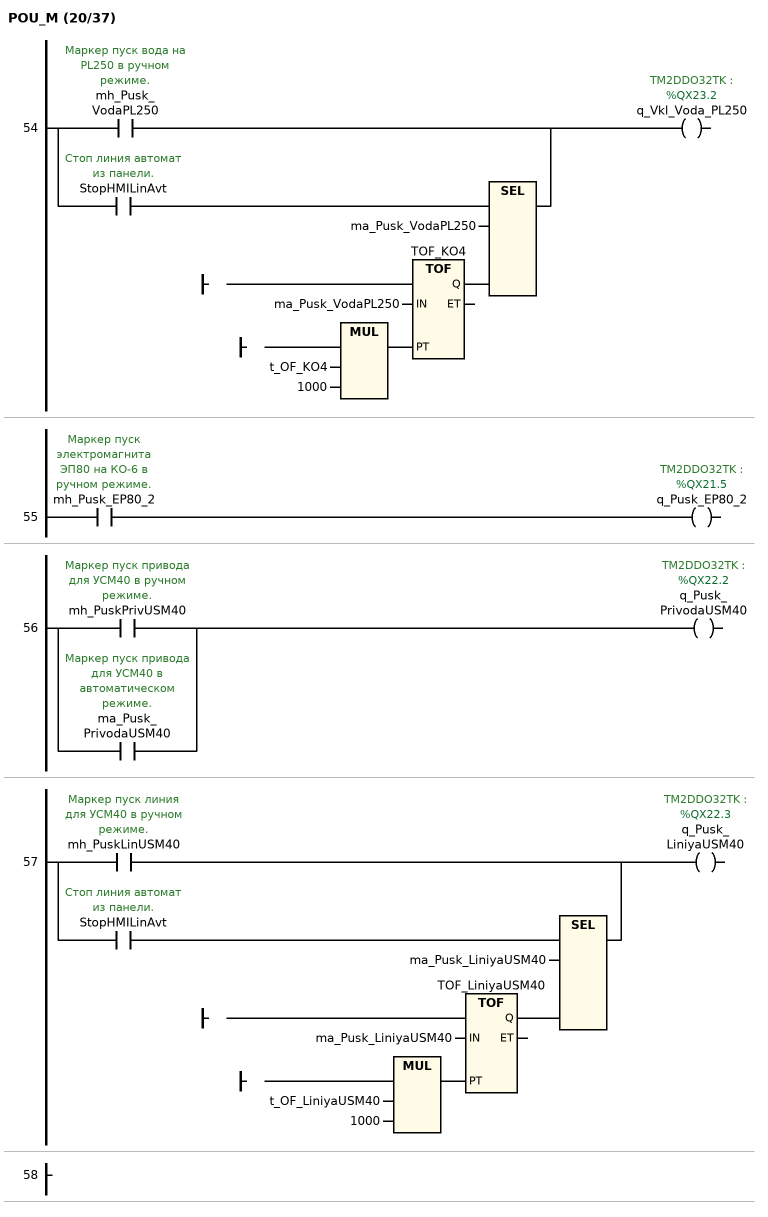
// NETWORK 54
//   mh_Pusk_VodaPL250: Маркер пуск вода на PL250 в ручном режиме.
//   StopHMILinAvt: Стоп линия автомат из панели.
//   ma_Pusk_VodaPL250: Маркер включение воды в питатель PL250 в автоматическом режиме.
//   TOF_KO4: Задержка перед выключением КО-4 при "Стоп линия автомат".
//   t_OF_KO4: Время задержки перед выключением КО-4 при Стоп Линия Автомат.
//   q_Vkl_Voda_PL250: TM2DDO32TK : | AT %QX23.2
TOF_KO4(IN := ma_Pusk_VodaPL250, PT := t_OF_KO4 * 1000); // TOF
q_Vkl_Voda_PL250 := mh_Pusk_VodaPL250 OR SEL(StopHMILinAvt, ma_Pusk_VodaPL250, TOF_KO4.Q);

// NETWORK 55
//   mh_Pusk_EP80_2: Маркер пуск электромагнита ЭП80 на КО-6 в ручном режиме.
//   q_Pusk_EP80_2: TM2DDO32TK : | AT %QX21.5
q_Pusk_EP80_2 := mh_Pusk_EP80_2;

// NETWORK 56
//   mh_PuskPrivUSM40: Маркер пуск привода для УСМ40 в ручном режиме.
//   ma_Pusk_PrivodaUSM40: Маркер пуск привода для УСМ40 в автоматическом режиме.
//   q_Pusk_PrivodaUSM40: TM2DDO32TK : | AT %QX22.2
q_Pusk_PrivodaUSM40 := mh_PuskPrivUSM40 OR ma_Pusk_PrivodaUSM40;

// NETWORK 57
//   mh_PuskLinUSM40: Маркер пуск линия для УСМ40 в ручном режиме.
//   StopHMILinAvt: Стоп линия автомат из панели.
//   ma_Pusk_LiniyaUSM40: Маркер пуск линия для УСМ40 в автоматическом режиме.
//   TOF_LiniyaUSM40: Задержка перед выключением конвейера на УСМ40 при "Стоп линия автомат".
//   t_OF_LiniyaUSM40: Время задержки перед выключением линии на УСМ40 при Стоп Линия Автомат.
//   q_Pusk_LiniyaUSM40: TM2DDO32TK : | AT %QX22.3
TOF_LiniyaUSM40(IN := ma_Pusk_LiniyaUSM40, PT := t_OF_LiniyaUSM40 * 1000); // TOF
q_Pusk_LiniyaUSM40 := mh_PuskLinUSM40 OR SEL(StopHMILinAvt, ma_Pusk_LiniyaUSM40, TOF_LiniyaUSM40.Q);

// NETWORK 58

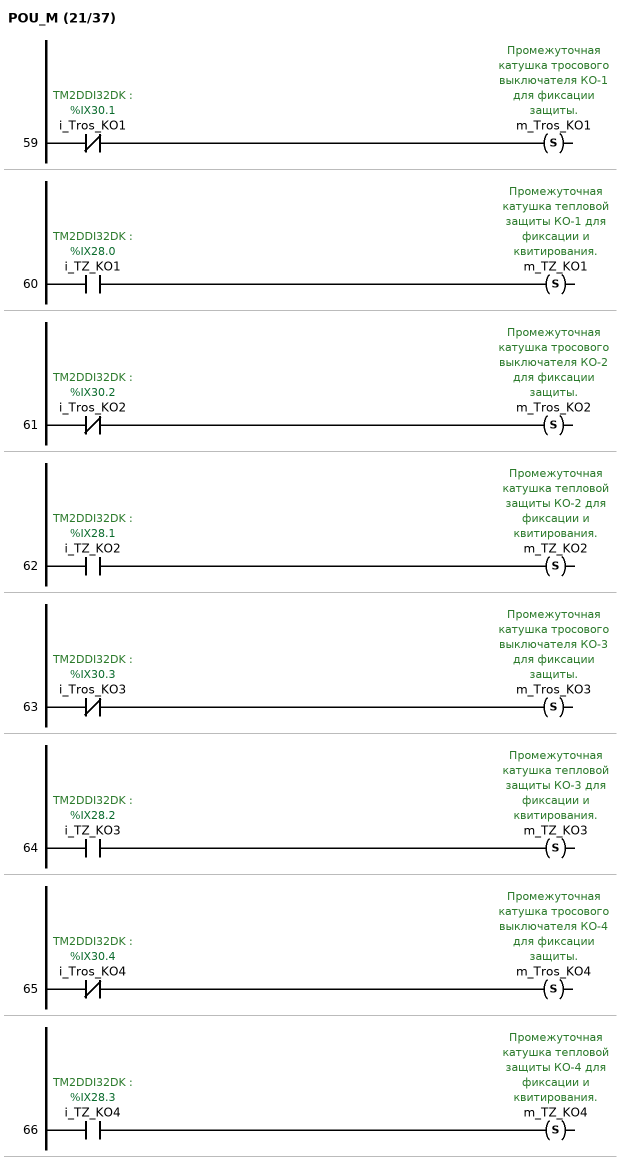
// NETWORK 59
//   i_Tros_KO1: TM2DDI32DK : | AT %IX30.1
//   m_Tros_KO1: Промежуточная катушка тросового выключателя КО-1 для фиксации защиты.
m_Tros_KO1 S= NOT i_Tros_KO1;

// NETWORK 60
//   i_TZ_KO1: TM2DDI32DK : | AT %IX28.0
//   m_TZ_KO1: Промежуточная катушка тепловой защиты КО-1 для фиксации и квитирования.
m_TZ_KO1 S= i_TZ_KO1;

// NETWORK 61
//   i_Tros_KO2: TM2DDI32DK : | AT %IX30.2
//   m_Tros_KO2: Промежуточная катушка тросового выключателя КО-2 для фиксации защиты.
m_Tros_KO2 S= NOT i_Tros_KO2;

// NETWORK 62
//   i_TZ_KO2: TM2DDI32DK : | AT %IX28.1
//   m_TZ_KO2: Промежуточная катушка тепловой защиты КО-2 для фиксации и квитирования.
m_TZ_KO2 S= i_TZ_KO2;

// NETWORK 63
//   i_Tros_KO3: TM2DDI32DK : | AT %IX30.3
//   m_Tros_KO3: Промежуточная катушка тросового выключателя КО-3 для фиксации защиты.
m_Tros_KO3 S= NOT i_Tros_KO3;

// NETWORK 64
//   i_TZ_KO3: TM2DDI32DK : | AT %IX28.2
//   m_TZ_KO3: Промежуточная катушка тепловой защиты КО-3 для фиксации и квитирования.
m_TZ_KO3 S= i_TZ_KO3;

// NETWORK 65
//   i_Tros_KO4: TM2DDI32DK : | AT %IX30.4
//   m_Tros_KO4: Промежуточная катушка тросового выключателя КО-4 для фиксации защиты.
m_Tros_KO4 S= NOT i_Tros_KO4;

// NETWORK 66
//   i_TZ_KO4: TM2DDI32DK : | AT %IX28.3
//   m_TZ_KO4: Промежуточная катушка тепловой защиты КО-4 для фиксации и квитирования.
m_TZ_KO4 S= i_TZ_KO4;

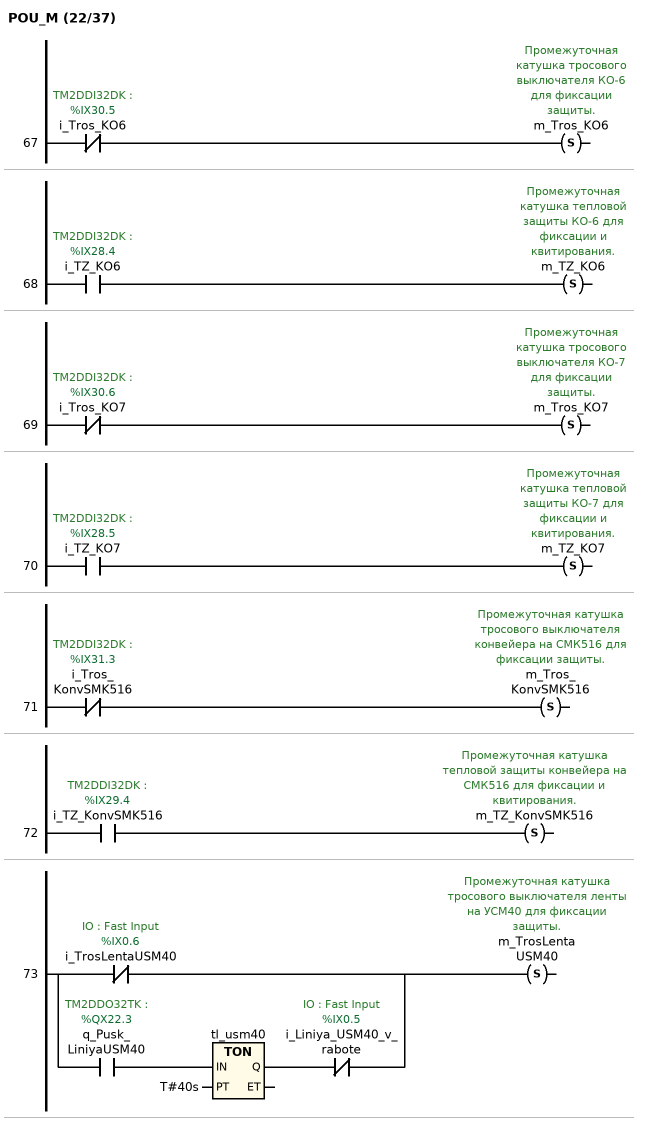
// NETWORK 67
//   i_Tros_KO6: TM2DDI32DK : | AT %IX30.5
//   m_Tros_KO6: Промежуточная катушка тросового выключателя КО-6 для фиксации защиты.
m_Tros_KO6 S= NOT i_Tros_KO6;

// NETWORK 68
//   i_TZ_KO6: TM2DDI32DK : | AT %IX28.4
//   m_TZ_KO6: Промежуточная катушка тепловой защиты КО-6 для фиксации и квитирования.
m_TZ_KO6 S= i_TZ_KO6;

// NETWORK 69
//   i_Tros_KO7: TM2DDI32DK : | AT %IX30.6
//   m_Tros_KO7: Промежуточная катушка тросового выключателя КО-7 для фиксации защиты.
m_Tros_KO7 S= NOT i_Tros_KO7;

// NETWORK 70
//   i_TZ_KO7: TM2DDI32DK : | AT %IX28.5
//   m_TZ_KO7: Промежуточная катушка тепловой защиты КО-7 для фиксации и квитирования.
m_TZ_KO7 S= i_TZ_KO7;

// NETWORK 71
//   i_Tros_KonvSMK516: TM2DDI32DK : | AT %IX31.3
//   m_Tros_KonvSMK516: Промежуточная катушка тросового выключателя конвейера на СМК516 для фиксации защиты.
m_Tros_KonvSMK516 S= NOT i_Tros_KonvSMK516;

// NETWORK 72
//   i_TZ_KonvSMK516: TM2DDI32DK : | AT %IX29.4
//   m_TZ_KonvSMK516: Промежуточная катушка тепловой защиты конвейера на СМК516 для фиксации и квитирования.
m_TZ_KonvSMK516 S= i_TZ_KonvSMK516;

// NETWORK 73
//   i_TrosLentaUSM40: IO : Fast Input | AT %IX0.6
//   q_Pusk_LiniyaUSM40: TM2DDO32TK : | AT %QX22.3
//   i_Liniya_USM40_v_rabote: IO : Fast Input | AT %IX0.5
//   m_TrosLentaUSM40: Промежуточная катушка тросового выключателя ленты на УСМ40 для фиксации защиты.
tl_usm40(IN := q_Pusk_LiniyaUSM40, PT := T#40s); // TON
m_TrosLentaUSM40 S= NOT i_TrosLentaUSM40 OR tl_usm40.Q AND NOT i_Liniya_USM40_v_rabote;

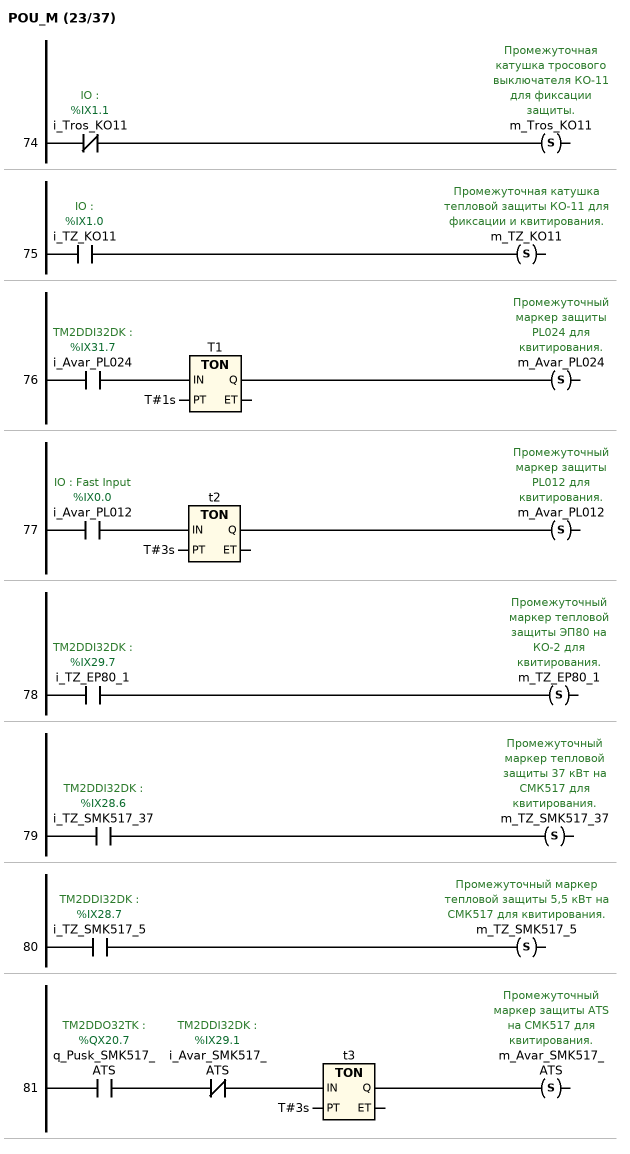
// NETWORK 74
//   i_Tros_KO11: IO : | AT %IX1.1
//   m_Tros_KO11: Промежуточная катушка тросового выключателя КО-11 для фиксации защиты.
m_Tros_KO11 S= NOT i_Tros_KO11;

// NETWORK 75
//   i_TZ_KO11: IO : | AT %IX1.0
//   m_TZ_KO11: Промежуточная катушка тепловой защиты КО-11 для фиксации и квитирования.
m_TZ_KO11 S= i_TZ_KO11;

// NETWORK 76
//   i_Avar_PL024: TM2DDI32DK : | AT %IX31.7
//   m_Avar_PL024: Промежуточный маркер защиты PL024 для квитирования.
T1(IN := i_Avar_PL024, PT := T#1s); // TON
m_Avar_PL024 S= T1.Q;

// NETWORK 77
//   i_Avar_PL012: IO : Fast Input | AT %IX0.0
//   m_Avar_PL012: Промежуточный маркер защиты PL012 для квитирования.
t2(IN := i_Avar_PL012, PT := T#3s); // TON
m_Avar_PL012 S= t2.Q;

// NETWORK 78
//   i_TZ_EP80_1: TM2DDI32DK : | AT %IX29.7
//   m_TZ_EP80_1: Промежуточный маркер тепловой защиты ЭП80 на КО-2 для квитирования.
m_TZ_EP80_1 S= i_TZ_EP80_1;

// NETWORK 79
//   i_TZ_SMK517_37: TM2DDI32DK : | AT %IX28.6
//   m_TZ_SMK517_37: Промежуточный маркер тепловой защиты 37 кВт на СМК517 для квитирования.
m_TZ_SMK517_37 S= i_TZ_SMK517_37;

// NETWORK 80
//   i_TZ_SMK517_5: TM2DDI32DK : | AT %IX28.7
//   m_TZ_SMK517_5: Промежуточный маркер тепловой защиты 5,5 кВт на СМК517 для квитирования.
m_TZ_SMK517_5 S= i_TZ_SMK517_5;

// NETWORK 81
//   q_Pusk_SMK517_ATS: TM2DDO32TK : | AT %QX20.7
//   i_Avar_SMK517_ATS: TM2DDI32DK : | AT %IX29.1
//   m_Avar_SMK517_ATS: Промежуточный маркер защиты ATS на СМК517 для квитирования.
t3(IN := q_Pusk_SMK517_ATS AND NOT i_Avar_SMK517_ATS, PT := T#3s); // TON
m_Avar_SMK517_ATS S= t3.Q;

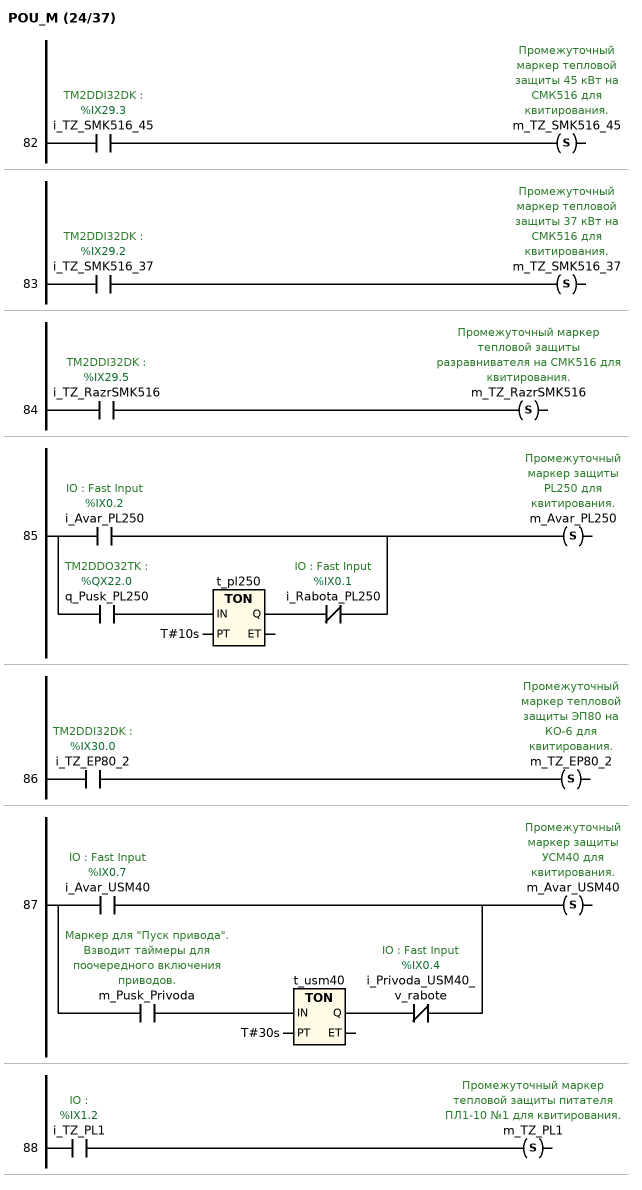
// NETWORK 82
//   i_TZ_SMK516_45: TM2DDI32DK : | AT %IX29.3
//   m_TZ_SMK516_45: Промежуточный маркер тепловой защиты 45 кВт на СМК516 для квитирования.
m_TZ_SMK516_45 S= i_TZ_SMK516_45;

// NETWORK 83
//   i_TZ_SMK516_37: TM2DDI32DK : | AT %IX29.2
//   m_TZ_SMK516_37: Промежуточный маркер тепловой защиты 37 кВт на СМК516 для квитирования.
m_TZ_SMK516_37 S= i_TZ_SMK516_37;

// NETWORK 84
//   i_TZ_RazrSMK516: TM2DDI32DK : | AT %IX29.5
//   m_TZ_RazrSMK516: Промежуточный маркер тепловой защиты разравнивателя на СМК516 для квитирования.
m_TZ_RazrSMK516 S= i_TZ_RazrSMK516;

// NETWORK 85
//   i_Avar_PL250: IO : Fast Input | AT %IX0.2
//   q_Pusk_PL250: TM2DDO32TK : | AT %QX22.0
//   i_Rabota_PL250: IO : Fast Input | AT %IX0.1
//   m_Avar_PL250: Промежуточный маркер защиты PL250 для квитирования.
t_pl250(IN := q_Pusk_PL250, PT := T#10s); // TON
m_Avar_PL250 S= i_Avar_PL250 OR t_pl250.Q AND NOT i_Rabota_PL250;

// NETWORK 86
//   i_TZ_EP80_2: TM2DDI32DK : | AT %IX30.0
//   m_TZ_EP80_2: Промежуточный маркер тепловой защиты ЭП80 на КО-6 для квитирования.
m_TZ_EP80_2 S= i_TZ_EP80_2;

// NETWORK 87
//   i_Avar_USM40: IO : Fast Input | AT %IX0.7
//   m_Pusk_Privoda: Маркер для "Пуск привода". Взводит таймеры для поочередного включения приводов.
//   i_Privoda_USM40_v_rabote: IO : Fast Input | AT %IX0.4
//   m_Avar_USM40: Промежуточный маркер защиты УСМ40 для квитирования.
t_usm40(IN := m_Pusk_Privoda, PT := T#30s); // TON
m_Avar_USM40 S= i_Avar_USM40 OR t_usm40.Q AND NOT i_Privoda_USM40_v_rabote;

// NETWORK 88
//   i_TZ_PL1: IO : | AT %IX1.2
//   m_TZ_PL1: Промежуточный маркер тепловой защиты питателя ПЛ1-10 №1 для квитирования.
m_TZ_PL1 S= i_TZ_PL1;

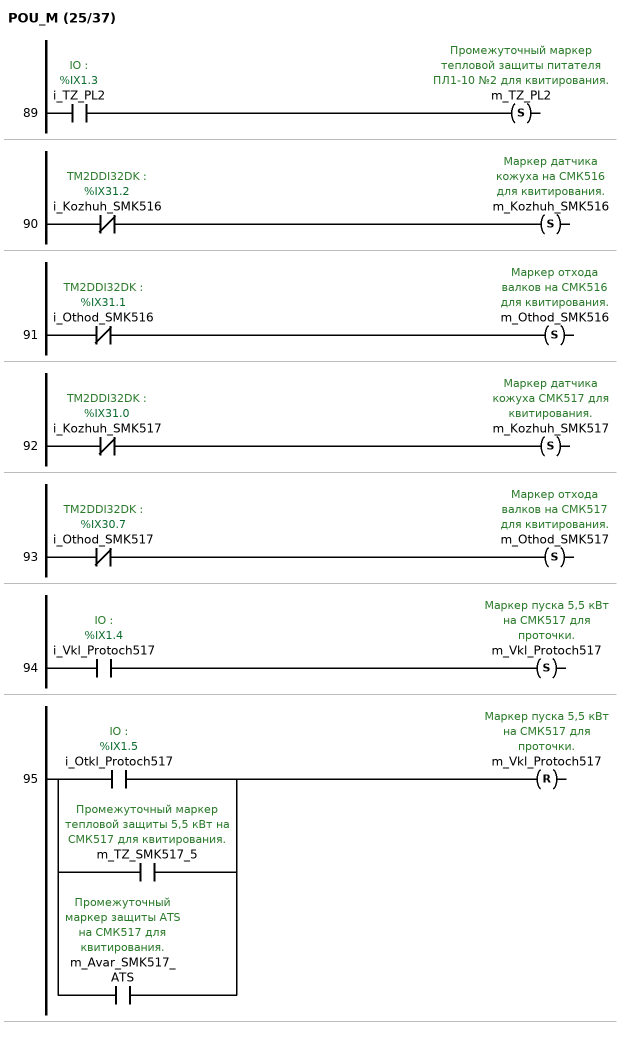
// NETWORK 89
//   i_TZ_PL2: IO : | AT %IX1.3
//   m_TZ_PL2: Промежуточный маркер тепловой защиты питателя ПЛ1-10 №2 для квитирования.
m_TZ_PL2 S= i_TZ_PL2;

// NETWORK 90
//   i_Kozhuh_SMK516: TM2DDI32DK : | AT %IX31.2
//   m_Kozhuh_SMK516: Маркер датчика кожуха на СМК516 для квитирования.
m_Kozhuh_SMK516 S= NOT i_Kozhuh_SMK516;

// NETWORK 91
//   i_Othod_SMK516: TM2DDI32DK : | AT %IX31.1
//   m_Othod_SMK516: Маркер отхода валков на СМК516 для квитирования.
m_Othod_SMK516 S= NOT i_Othod_SMK516;

// NETWORK 92
//   i_Kozhuh_SMK517: TM2DDI32DK : | AT %IX31.0
//   m_Kozhuh_SMK517: Маркер датчика кожуха СМК517 для квитирования.
m_Kozhuh_SMK517 S= NOT i_Kozhuh_SMK517;

// NETWORK 93
//   i_Othod_SMK517: TM2DDI32DK : | AT %IX30.7
//   m_Othod_SMK517: Маркер отхода валков на СМК517 для квитирования.
m_Othod_SMK517 S= NOT i_Othod_SMK517;

// NETWORK 94
//   i_Vkl_Protoch517: IO : | AT %IX1.4
//   m_Vkl_Protoch517: Маркер пуска 5,5 кВт на СМК517 для проточки.
m_Vkl_Protoch517 S= i_Vkl_Protoch517;

// NETWORK 95
//   i_Otkl_Protoch517: IO : | AT %IX1.5
//   m_TZ_SMK517_5: Промежуточный маркер тепловой защиты 5,5 кВт на СМК517 для квитирования.
//   m_Avar_SMK517_ATS: Промежуточный маркер защиты ATS на СМК517 для квитирования.
//   m_Vkl_Protoch517: Маркер пуска 5,5 кВт на СМК517 для проточки.
m_Vkl_Protoch517 R= i_Otkl_Protoch517 OR m_TZ_SMK517_5 OR m_Avar_SMK517_ATS;

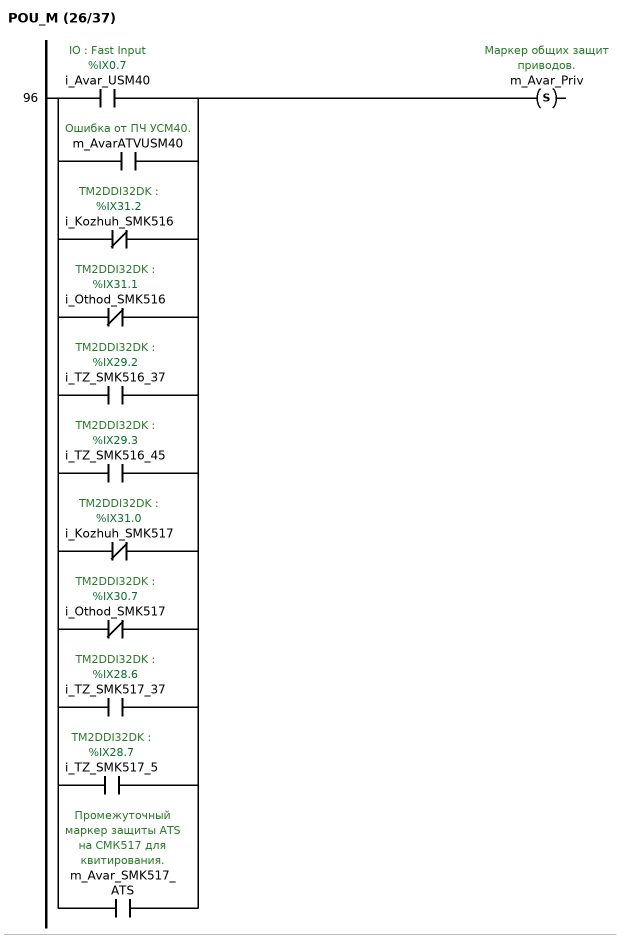
// NETWORK 96
//   i_Avar_USM40: IO : Fast Input | AT %IX0.7
//   m_AvarATVUSM40: Ошибка от ПЧ УСМ40.
//   i_Kozhuh_SMK516: TM2DDI32DK : | AT %IX31.2
//   i_Othod_SMK516: TM2DDI32DK : | AT %IX31.1
//   i_TZ_SMK516_37: TM2DDI32DK : | AT %IX29.2
//   i_TZ_SMK516_45: TM2DDI32DK : | AT %IX29.3
//   i_Kozhuh_SMK517: TM2DDI32DK : | AT %IX31.0
//   i_Othod_SMK517: TM2DDI32DK : | AT %IX30.7
//   i_TZ_SMK517_37: TM2DDI32DK : | AT %IX28.6
//   i_TZ_SMK517_5: TM2DDI32DK : | AT %IX28.7
//   m_Avar_SMK517_ATS: Промежуточный маркер защиты ATS на СМК517 для квитирования.
//   m_Avar_Priv: Маркер общих защит приводов.
m_Avar_Priv S= i_Avar_USM40 OR m_AvarATVUSM40 OR NOT i_Kozhuh_SMK516 OR NOT i_Othod_SMK516 OR i_TZ_SMK516_37 OR i_TZ_SMK516_45 OR NOT i_Kozhuh_SMK517 OR NOT i_Othod_SMK517 OR i_TZ_SMK517_37 OR i_TZ_SMK517_5 OR m_Avar_SMK517_ATS;

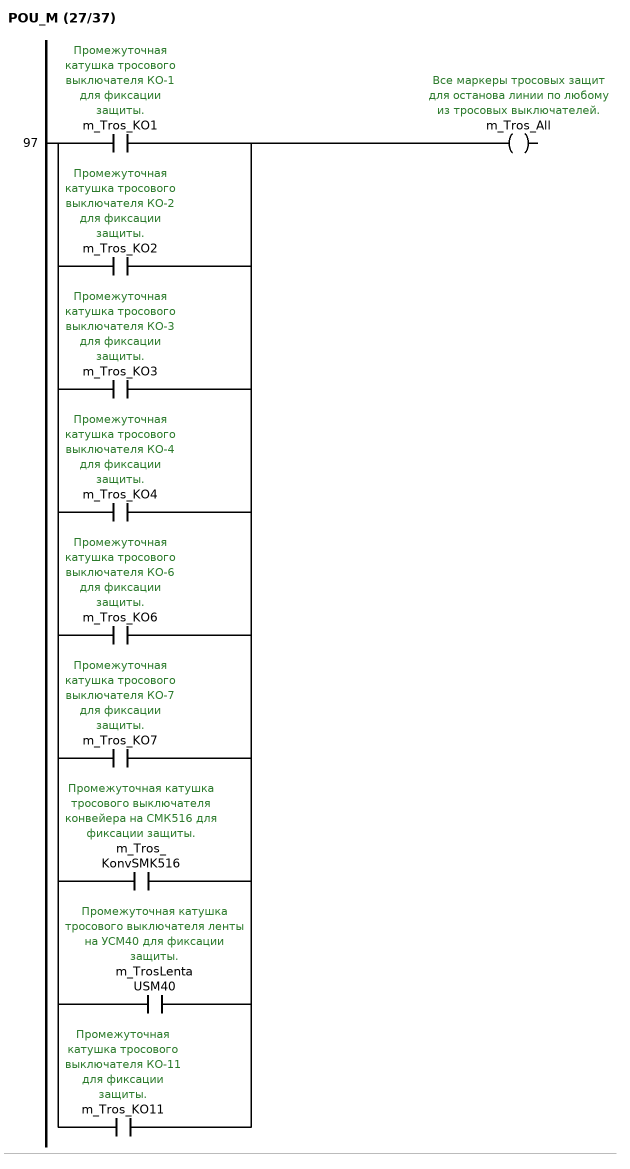
// NETWORK 97
//   m_Tros_KO1: Промежуточная катушка тросового выключателя КО-1 для фиксации защиты.
//   m_Tros_KO2: Промежуточная катушка тросового выключателя КО-2 для фиксации защиты.
//   m_Tros_KO3: Промежуточная катушка тросового выключателя КО-3 для фиксации защиты.
//   m_Tros_KO4: Промежуточная катушка тросового выключателя КО-4 для фиксации защиты.
//   m_Tros_KO6: Промежуточная катушка тросового выключателя КО-6 для фиксации защиты.
//   m_Tros_KO7: Промежуточная катушка тросового выключателя КО-7 для фиксации защиты.
//   m_Tros_KonvSMK516: Промежуточная катушка тросового выключателя конвейера на СМК516 для фиксации защиты.
//   m_TrosLentaUSM40: Промежуточная катушка тросового выключателя ленты на УСМ40 для фиксации защиты.
//   m_Tros_KO11: Промежуточная катушка тросового выключателя КО-11 для фиксации защиты.
//   m_Tros_All: Все маркеры тросовых защит для останова линии по любому из тросовых выключателей.
m_Tros_All := m_Tros_KO1 OR m_Tros_KO2 OR m_Tros_KO3 OR m_Tros_KO4 OR m_Tros_KO6 OR m_Tros_KO7 OR m_Tros_KonvSMK516 OR m_TrosLentaUSM40 OR m_Tros_KO11;

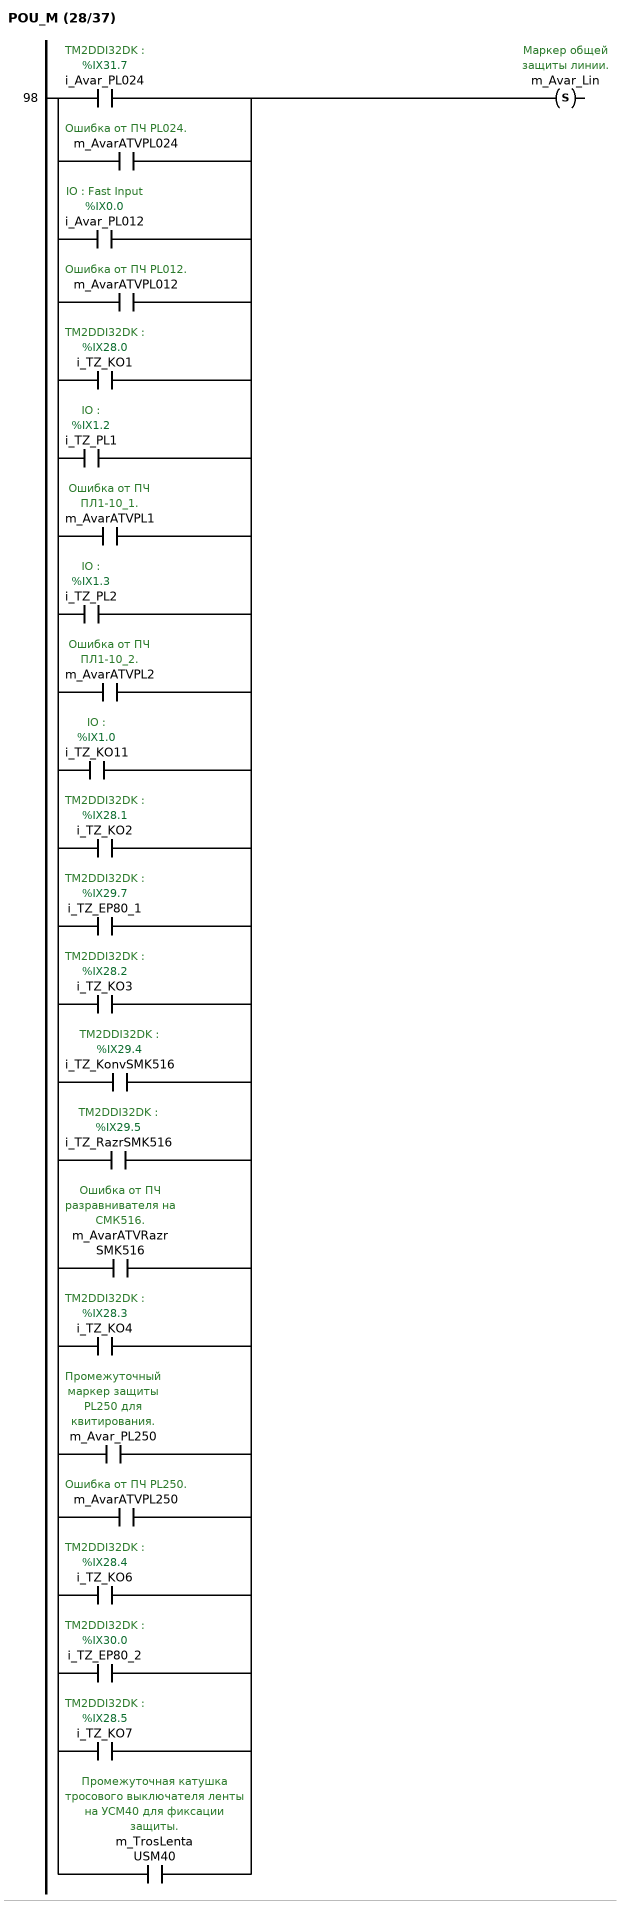
// NETWORK 98
//   i_Avar_PL024: TM2DDI32DK : | AT %IX31.7
//   m_AvarATVPL024: Ошибка от ПЧ PL024.
//   i_Avar_PL012: IO : Fast Input | AT %IX0.0
//   m_AvarATVPL012: Ошибка от ПЧ PL012.
//   i_TZ_KO1: TM2DDI32DK : | AT %IX28.0
//   i_TZ_PL1: IO : | AT %IX1.2
//   m_AvarATVPL1: Ошибка от ПЧ ПЛ1-10_1.
//   i_TZ_PL2: IO : | AT %IX1.3
//   m_AvarATVPL2: Ошибка от ПЧ ПЛ1-10_2.
//   i_TZ_KO11: IO : | AT %IX1.0
//   i_TZ_KO2: TM2DDI32DK : | AT %IX28.1
//   i_TZ_EP80_1: TM2DDI32DK : | AT %IX29.7
//   i_TZ_KO3: TM2DDI32DK : | AT %IX28.2
//   i_TZ_KonvSMK516: TM2DDI32DK : | AT %IX29.4
//   i_TZ_RazrSMK516: TM2DDI32DK : | AT %IX29.5
//   m_AvarATVRazrSMK516: Ошибка от ПЧ разравнивателя на СМК516.
//   i_TZ_KO4: TM2DDI32DK : | AT %IX28.3
//   m_Avar_PL250: Промежуточный маркер защиты PL250 для квитирования.
//   m_AvarATVPL250: Ошибка от ПЧ PL250.
//   i_TZ_KO6: TM2DDI32DK : | AT %IX28.4
//   i_TZ_EP80_2: TM2DDI32DK : | AT %IX30.0
//   i_TZ_KO7: TM2DDI32DK : | AT %IX28.5
//   m_TrosLentaUSM40: Промежуточная катушка тросового выключателя ленты на УСМ40 для фиксации защиты.
//   m_Avar_Lin: Маркер общей защиты линии.
m_Avar_Lin S= i_Avar_PL024 OR m_AvarATVPL024 OR i_Avar_PL012 OR m_AvarATVPL012 OR i_TZ_KO1 OR i_TZ_PL1 OR m_AvarATVPL1 OR i_TZ_PL2 OR m_AvarATVPL2 OR i_TZ_KO11 OR i_TZ_KO2 OR i_TZ_EP80_1 OR i_TZ_KO3 OR i_TZ_KonvSMK516 OR i_TZ_RazrSMK516 OR m_AvarATVRazrSMK516 OR i_TZ_KO4 OR m_Avar_PL250 OR m_AvarATVPL250 OR i_TZ_KO6 OR i_TZ_EP80_2 OR i_TZ_KO7 OR m_TrosLentaUSM40;

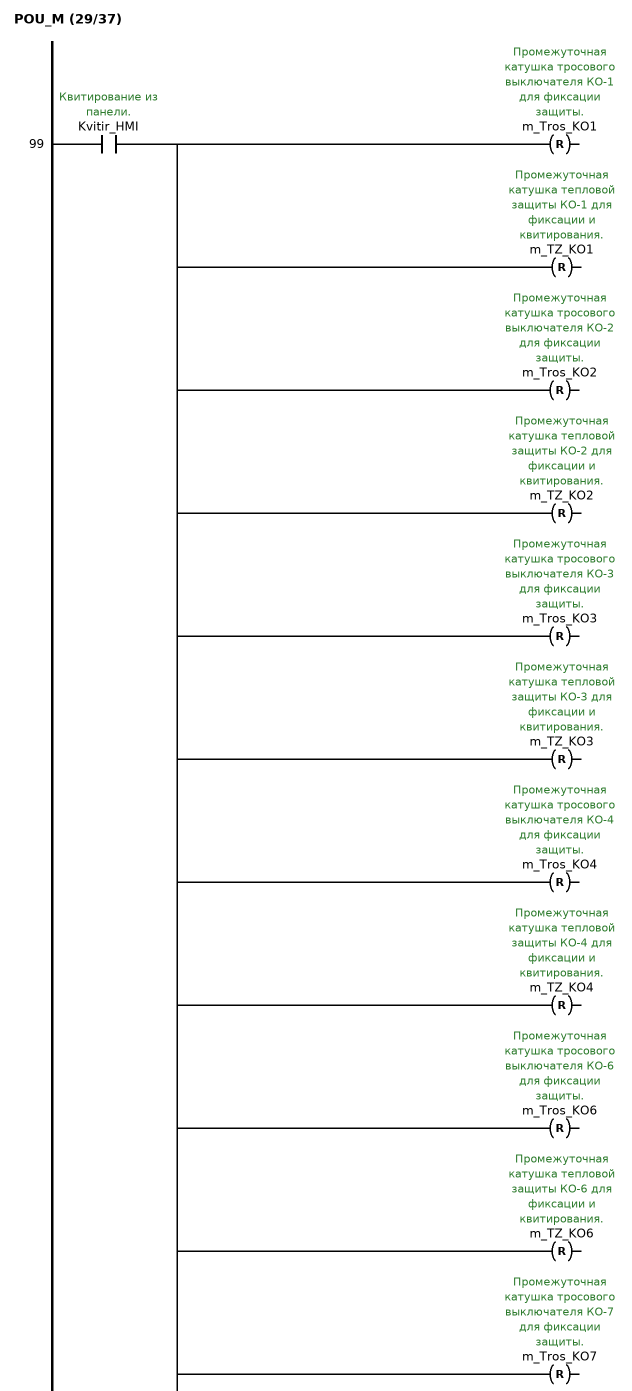
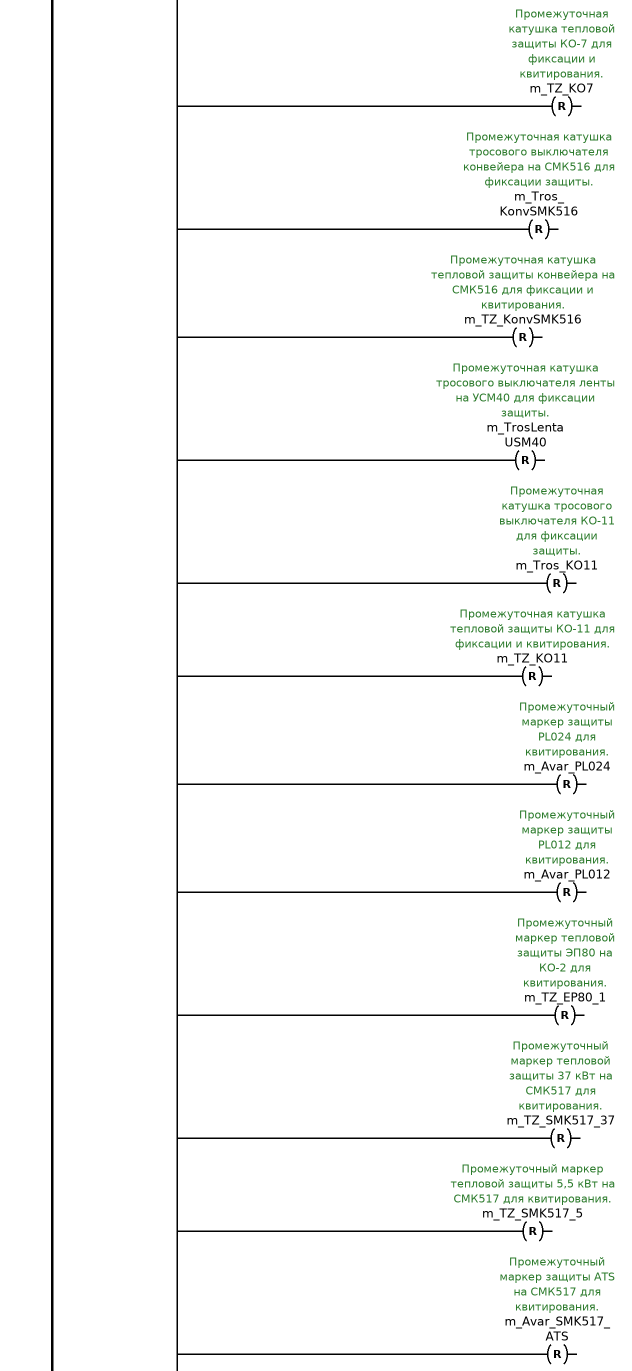
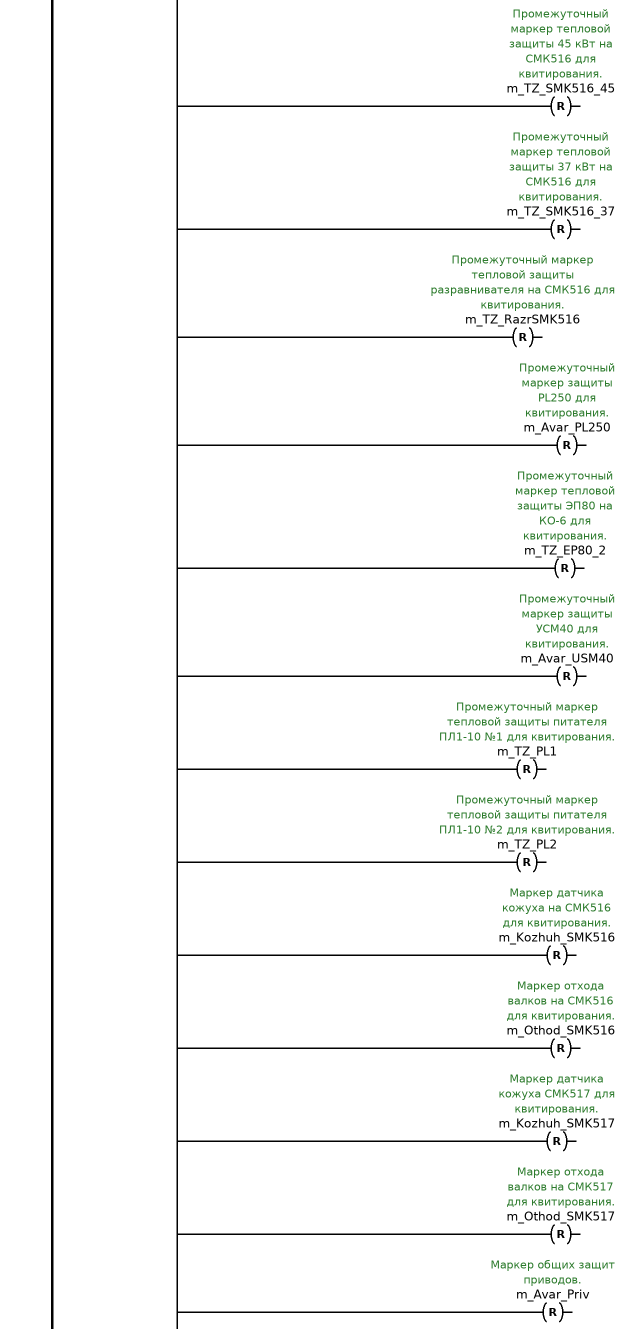
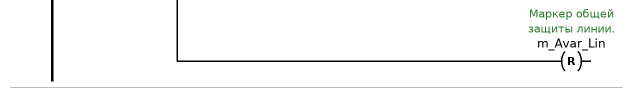
// NETWORK 99
//   Kvitir_HMI: Квитирование из панели.
//   m_Tros_KO1: Промежуточная катушка тросового выключателя КО-1 для фиксации защиты.
//   m_TZ_KO1: Промежуточная катушка тепловой защиты КО-1 для фиксации и квитирования.
//   m_Tros_KO2: Промежуточная катушка тросового выключателя КО-2 для фиксации защиты.
//   m_TZ_KO2: Промежуточная катушка тепловой защиты КО-2 для фиксации и квитирования.
//   m_Tros_KO3: Промежуточная катушка тросового выключателя КО-3 для фиксации защиты.
//   m_TZ_KO3: Промежуточная катушка тепловой защиты КО-3 для фиксации и квитирования.
//   m_Tros_KO4: Промежуточная катушка тросового выключателя КО-4 для фиксации защиты.
//   m_TZ_KO4: Промежуточная катушка тепловой защиты КО-4 для фиксации и квитирования.
//   m_Tros_KO6: Промежуточная катушка тросового выключателя КО-6 для фиксации защиты.
//   m_TZ_KO6: Промежуточная катушка тепловой защиты КО-6 для фиксации и квитирования.
//   m_Tros_KO7: Промежуточная катушка тросового выключателя КО-7 для фиксации защиты.
//   m_TZ_KO7: Промежуточная катушка тепловой защиты КО-7 для фиксации и квитирования.
//   m_Tros_KonvSMK516: Промежуточная катушка тросового выключателя конвейера на СМК516 для фиксации защиты.
//   m_TZ_KonvSMK516: Промежуточная катушка тепловой защиты конвейера на СМК516 для фиксации и квитирования.
//   m_TrosLentaUSM40: Промежуточная катушка тросового выключателя ленты на УСМ40 для фиксации защиты.
//   m_Tros_KO11: Промежуточная катушка тросового выключателя КО-11 для фиксации защиты.
//   m_TZ_KO11: Промежуточная катушка тепловой защиты КО-11 для фиксации и квитирования.
//   m_Avar_PL024: Промежуточный маркер защиты PL024 для квитирования.
//   m_Avar_PL012: Промежуточный маркер защиты PL012 для квитирования.
//   m_TZ_EP80_1: Промежуточный маркер тепловой защиты ЭП80 на КО-2 для квитирования.
//   m_TZ_SMK517_37: Промежуточный маркер тепловой защиты 37 кВт на СМК517 для квитирования.
//   m_TZ_SMK517_5: Промежуточный маркер тепловой защиты 5,5 кВт на СМК517 для квитирования.
//   m_Avar_SMK517_ATS: Промежуточный маркер защиты ATS на СМК517 для квитирования.
//   m_TZ_SMK516_45: Промежуточный маркер тепловой защиты 45 кВт на СМК516 для квитирования.
//   m_TZ_SMK516_37: Промежуточный маркер тепловой защиты 37 кВт на СМК516 для квитирования.
//   m_TZ_RazrSMK516: Промежуточный маркер тепловой защиты разравнивателя на СМК516 для квитирования.
//   m_Avar_PL250: Промежуточный маркер защиты PL250 для квитирования.
//   m_TZ_EP80_2: Промежуточный маркер тепловой защиты ЭП80 на КО-6 для квитирования.
//   m_Avar_USM40: Промежуточный маркер защиты УСМ40 для квитирования.
//   m_TZ_PL1: Промежуточный маркер тепловой защиты питателя ПЛ1-10 №1 для квитирования.
//   m_TZ_PL2: Промежуточный маркер тепловой защиты питателя ПЛ1-10 №2 для квитирования.
//   m_Kozhuh_SMK516: Маркер датчика кожуха на СМК516 для квитирования.
//   m_Othod_SMK516: Маркер отхода валков на СМК516 для квитирования.
//   m_Kozhuh_SMK517: Маркер датчика кожуха СМК517 для квитирования.
//   m_Othod_SMK517: Маркер отхода валков на СМК517 для квитирования.
//   m_Avar_Priv: Маркер общих защит приводов.
//   m_Avar_Lin: Маркер общей защиты линии.
m_Tros_KO1 R= Kvitir_HMI;
m_TZ_KO1 R= Kvitir_HMI;
m_Tros_KO2 R= Kvitir_HMI;
m_TZ_KO2 R= Kvitir_HMI;
m_Tros_KO3 R= Kvitir_HMI;
m_TZ_KO3 R= Kvitir_HMI;
m_Tros_KO4 R= Kvitir_HMI;
m_TZ_KO4 R= Kvitir_HMI;
m_Tros_KO6 R= Kvitir_HMI;
m_TZ_KO6 R= Kvitir_HMI;
m_Tros_KO7 R= Kvitir_HMI;
m_TZ_KO7 R= Kvitir_HMI;
m_Tros_KonvSMK516 R= Kvitir_HMI;
m_TZ_KonvSMK516 R= Kvitir_HMI;
m_TrosLentaUSM40 R= Kvitir_HMI;
m_Tros_KO11 R= Kvitir_HMI;
m_TZ_KO11 R= Kvitir_HMI;
m_Avar_PL024 R= Kvitir_HMI;
m_Avar_PL012 R= Kvitir_HMI;
m_TZ_EP80_1 R= Kvitir_HMI;
m_TZ_SMK517_37 R= Kvitir_HMI;
m_TZ_SMK517_5 R= Kvitir_HMI;
m_Avar_SMK517_ATS R= Kvitir_HMI;
m_TZ_SMK516_45 R= Kvitir_HMI;
m_TZ_SMK516_37 R= Kvitir_HMI;
m_TZ_RazrSMK516 R= Kvitir_HMI;
m_Avar_PL250 R= Kvitir_HMI;
m_TZ_EP80_2 R= Kvitir_HMI;
m_Avar_USM40 R= Kvitir_HMI;
m_TZ_PL1 R= Kvitir_HMI;
m_TZ_PL2 R= Kvitir_HMI;
m_Kozhuh_SMK516 R= Kvitir_HMI;
m_Othod_SMK516 R= Kvitir_HMI;
m_Kozhuh_SMK517 R= Kvitir_HMI;
m_Othod_SMK517 R= Kvitir_HMI;
m_Avar_Priv R= Kvitir_HMI;
m_Avar_Lin R= Kvitir_HMI;

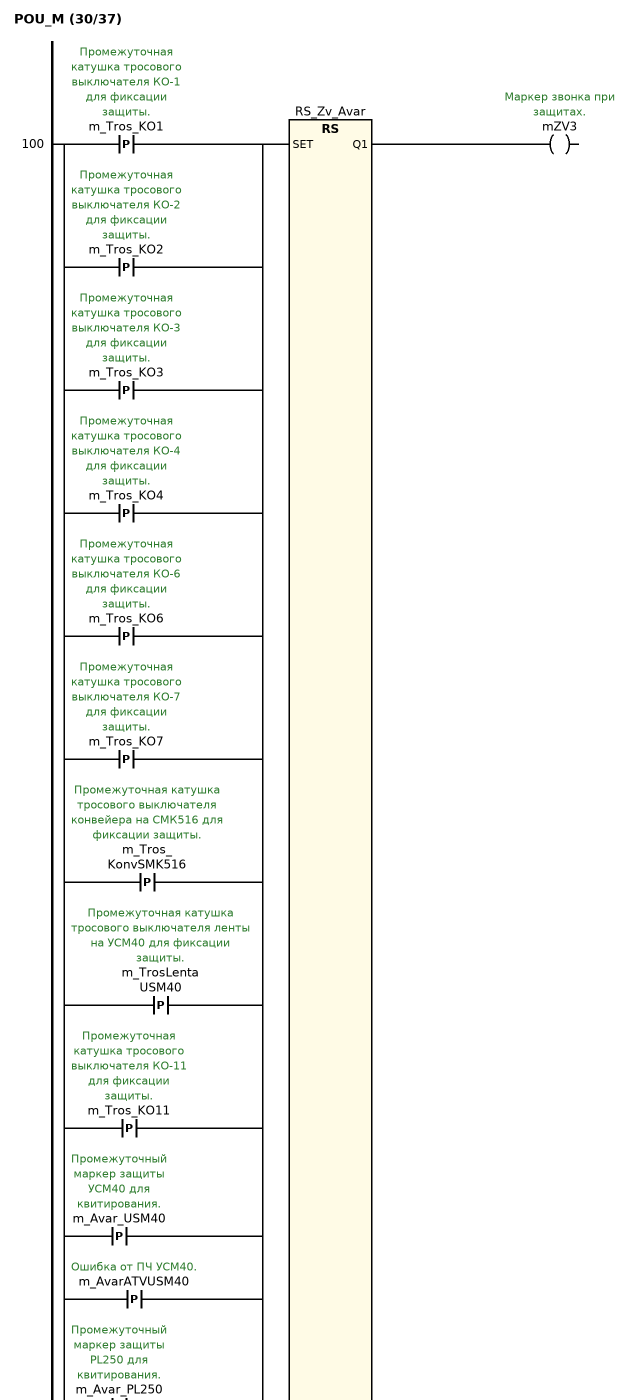
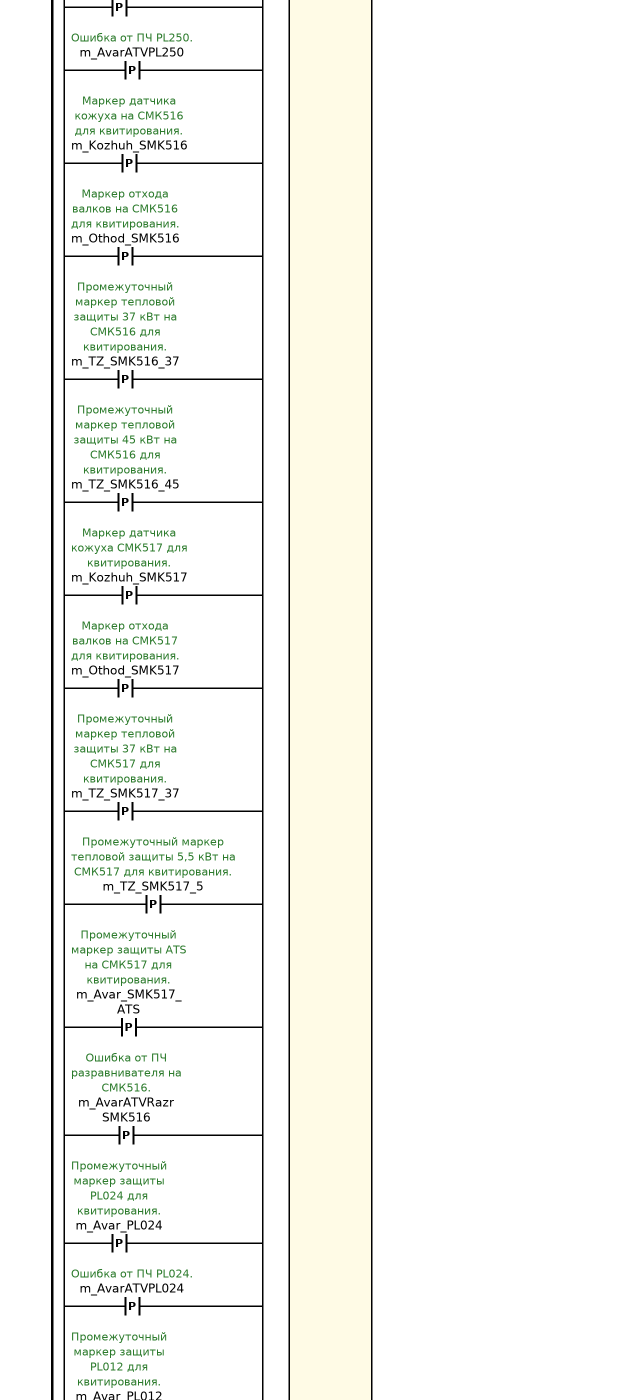
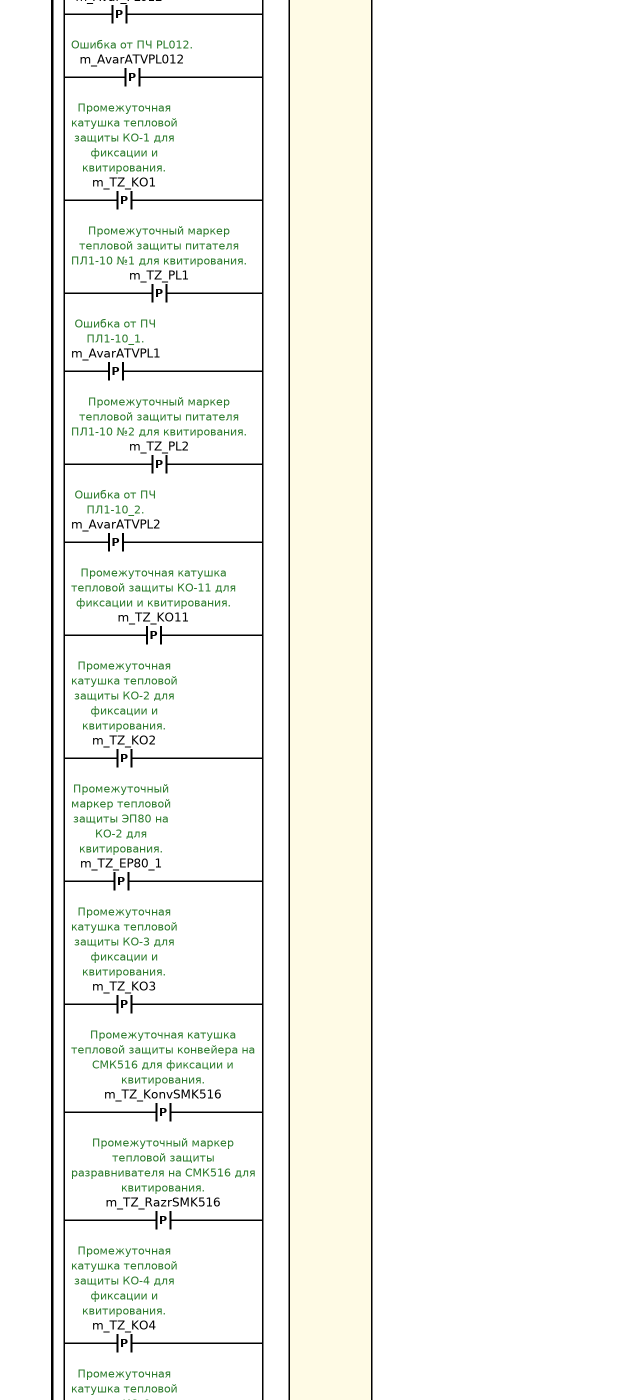
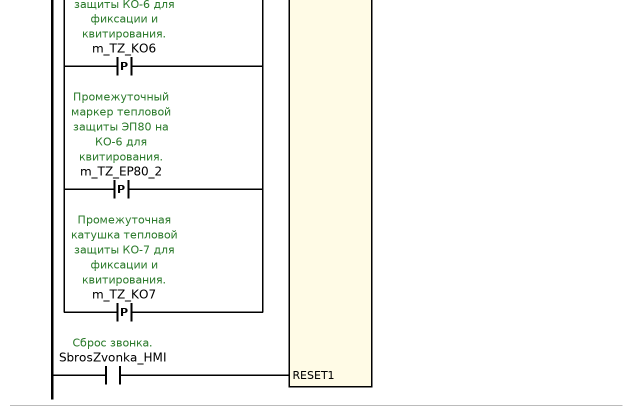
// NETWORK 100
//   RS_Zv_Avar: Триггер звонков при срабатывании защит.
//   m_Tros_KO1: Промежуточная катушка тросового выключателя КО-1 для фиксации защиты.
//   m_Tros_KO2: Промежуточная катушка тросового выключателя КО-2 для фиксации защиты.
//   m_Tros_KO3: Промежуточная катушка тросового выключателя КО-3 для фиксации защиты.
//   m_Tros_KO4: Промежуточная катушка тросового выключателя КО-4 для фиксации защиты.
//   m_Tros_KO6: Промежуточная катушка тросового выключателя КО-6 для фиксации защиты.
//   m_Tros_KO7: Промежуточная катушка тросового выключателя КО-7 для фиксации защиты.
//   m_Tros_KonvSMK516: Промежуточная катушка тросового выключателя конвейера на СМК516 для фиксации защиты.
//   m_TrosLentaUSM40: Промежуточная катушка тросового выключателя ленты на УСМ40 для фиксации защиты.
//   m_Tros_KO11: Промежуточная катушка тросового выключателя КО-11 для фиксации защиты.
//   m_Avar_USM40: Промежуточный маркер защиты УСМ40 для квитирования.
//   m_AvarATVUSM40: Ошибка от ПЧ УСМ40.
//   m_Avar_PL250: Промежуточный маркер защиты PL250 для квитирования.
//   m_AvarATVPL250: Ошибка от ПЧ PL250.
//   m_Kozhuh_SMK516: Маркер датчика кожуха на СМК516 для квитирования.
//   m_Othod_SMK516: Маркер отхода валков на СМК516 для квитирования.
//   m_TZ_SMK516_37: Промежуточный маркер тепловой защиты 37 кВт на СМК516 для квитирования.
//   m_TZ_SMK516_45: Промежуточный маркер тепловой защиты 45 кВт на СМК516 для квитирования.
//   m_Kozhuh_SMK517: Маркер датчика кожуха СМК517 для квитирования.
//   m_Othod_SMK517: Маркер отхода валков на СМК517 для квитирования.
//   m_TZ_SMK517_37: Промежуточный маркер тепловой защиты 37 кВт на СМК517 для квитирования.
//   m_TZ_SMK517_5: Промежуточный маркер тепловой защиты 5,5 кВт на СМК517 для квитирования.
//   m_Avar_SMK517_ATS: Промежуточный маркер защиты ATS на СМК517 для квитирования.
//   m_AvarATVRazrSMK516: Ошибка от ПЧ разравнивателя на СМК516.
//   m_Avar_PL024: Промежуточный маркер защиты PL024 для квитирования.
//   m_AvarATVPL024: Ошибка от ПЧ PL024.
//   m_Avar_PL012: Промежуточный маркер защиты PL012 для квитирования.
//   m_AvarATVPL012: Ошибка от ПЧ PL012.
//   m_TZ_KO1: Промежуточная катушка тепловой защиты КО-1 для фиксации и квитирования.
//   m_TZ_PL1: Промежуточный маркер тепловой защиты питателя ПЛ1-10 №1 для квитирования.
//   m_AvarATVPL1: Ошибка от ПЧ ПЛ1-10_1.
//   m_TZ_PL2: Промежуточный маркер тепловой защиты питателя ПЛ1-10 №2 для квитирования.
//   m_AvarATVPL2: Ошибка от ПЧ ПЛ1-10_2.
//   m_TZ_KO11: Промежуточная катушка тепловой защиты КО-11 для фиксации и квитирования.
//   m_TZ_KO2: Промежуточная катушка тепловой защиты КО-2 для фиксации и квитирования.
//   m_TZ_EP80_1: Промежуточный маркер тепловой защиты ЭП80 на КО-2 для квитирования.
//   m_TZ_KO3: Промежуточная катушка тепловой защиты КО-3 для фиксации и квитирования.
//   m_TZ_KonvSMK516: Промежуточная катушка тепловой защиты конвейера на СМК516 для фиксации и квитирования.
//   m_TZ_RazrSMK516: Промежуточный маркер тепловой защиты разравнивателя на СМК516 для квитирования.
//   m_TZ_KO4: Промежуточная катушка тепловой защиты КО-4 для фиксации и квитирования.
//   m_TZ_KO6: Промежуточная катушка тепловой защиты КО-6 для фиксации и квитирования.
//   m_TZ_EP80_2: Промежуточный маркер тепловой защиты ЭП80 на КО-6 для квитирования.
//   m_TZ_KO7: Промежуточная катушка тепловой защиты КО-7 для фиксации и квитирования.
//   SbrosZvonka_HMI: Сброс звонка.
//   mZV3: Маркер звонка при защитах.
_rt27(CLK := m_Tros_KO1);
_rt28(CLK := m_Tros_KO2);
_rt29(CLK := m_Tros_KO3);
_rt30(CLK := m_Tros_KO4);
_rt31(CLK := m_Tros_KO6);
_rt32(CLK := m_Tros_KO7);
_rt33(CLK := m_Tros_KonvSMK516);
_rt34(CLK := m_TrosLentaUSM40);
_rt35(CLK := m_Tros_KO11);
_rt36(CLK := m_Avar_USM40);
_rt37(CLK := m_AvarATVUSM40);
_rt38(CLK := m_Avar_PL250);
_rt39(CLK := m_AvarATVPL250);
_rt40(CLK := m_Kozhuh_SMK516);
_rt41(CLK := m_Othod_SMK516);
_rt42(CLK := m_TZ_SMK516_37);
_rt43(CLK := m_TZ_SMK516_45);
_rt44(CLK := m_Kozhuh_SMK517);
_rt45(CLK := m_Othod_SMK517);
_rt46(CLK := m_TZ_SMK517_37);
_rt47(CLK := m_TZ_SMK517_5);
_rt48(CLK := m_Avar_SMK517_ATS);
_rt49(CLK := m_AvarATVRazrSMK516);
_rt50(CLK := m_Avar_PL024);
_rt51(CLK := m_AvarATVPL024);
_rt52(CLK := m_Avar_PL012);
_rt53(CLK := m_AvarATVPL012);
_rt54(CLK := m_TZ_KO1);
_rt55(CLK := m_TZ_PL1);
_rt56(CLK := m_AvarATVPL1);
_rt57(CLK := m_TZ_PL2);
_rt58(CLK := m_AvarATVPL2);
_rt59(CLK := m_TZ_KO11);
_rt60(CLK := m_TZ_KO2);
_rt61(CLK := m_TZ_EP80_1);
_rt62(CLK := m_TZ_KO3);
_rt63(CLK := m_TZ_KonvSMK516);
_rt64(CLK := m_TZ_RazrSMK516);
_rt65(CLK := m_TZ_KO4);
_rt66(CLK := m_TZ_KO6);
_rt67(CLK := m_TZ_EP80_2);
_rt68(CLK := m_TZ_KO7);
RS_Zv_Avar(SET := _rt27.Q OR _rt28.Q OR _rt29.Q OR _rt30.Q OR _rt31.Q OR _rt32.Q OR _rt33.Q OR _rt34.Q OR _rt35.Q OR _rt36.Q OR _rt37.Q OR _rt38.Q OR _rt39.Q OR _rt40.Q OR _rt41.Q OR _rt42.Q OR _rt43.Q OR _rt44.Q OR _rt45.Q OR _rt46.Q OR _rt47.Q OR _rt48.Q OR _rt49.Q OR _rt50.Q OR _rt51.Q OR _rt52.Q OR _rt53.Q OR _rt54.Q OR _rt55.Q OR _rt56.Q OR _rt57.Q OR _rt58.Q OR _rt59.Q OR _rt60.Q OR _rt61.Q OR _rt62.Q OR _rt63.Q OR _rt64.Q OR _rt65.Q OR _rt66.Q OR _rt67.Q OR _rt68.Q, RESET1 := SbrosZvonka_HMI); // RS
mZV3 := RS_Zv_Avar.Q1;

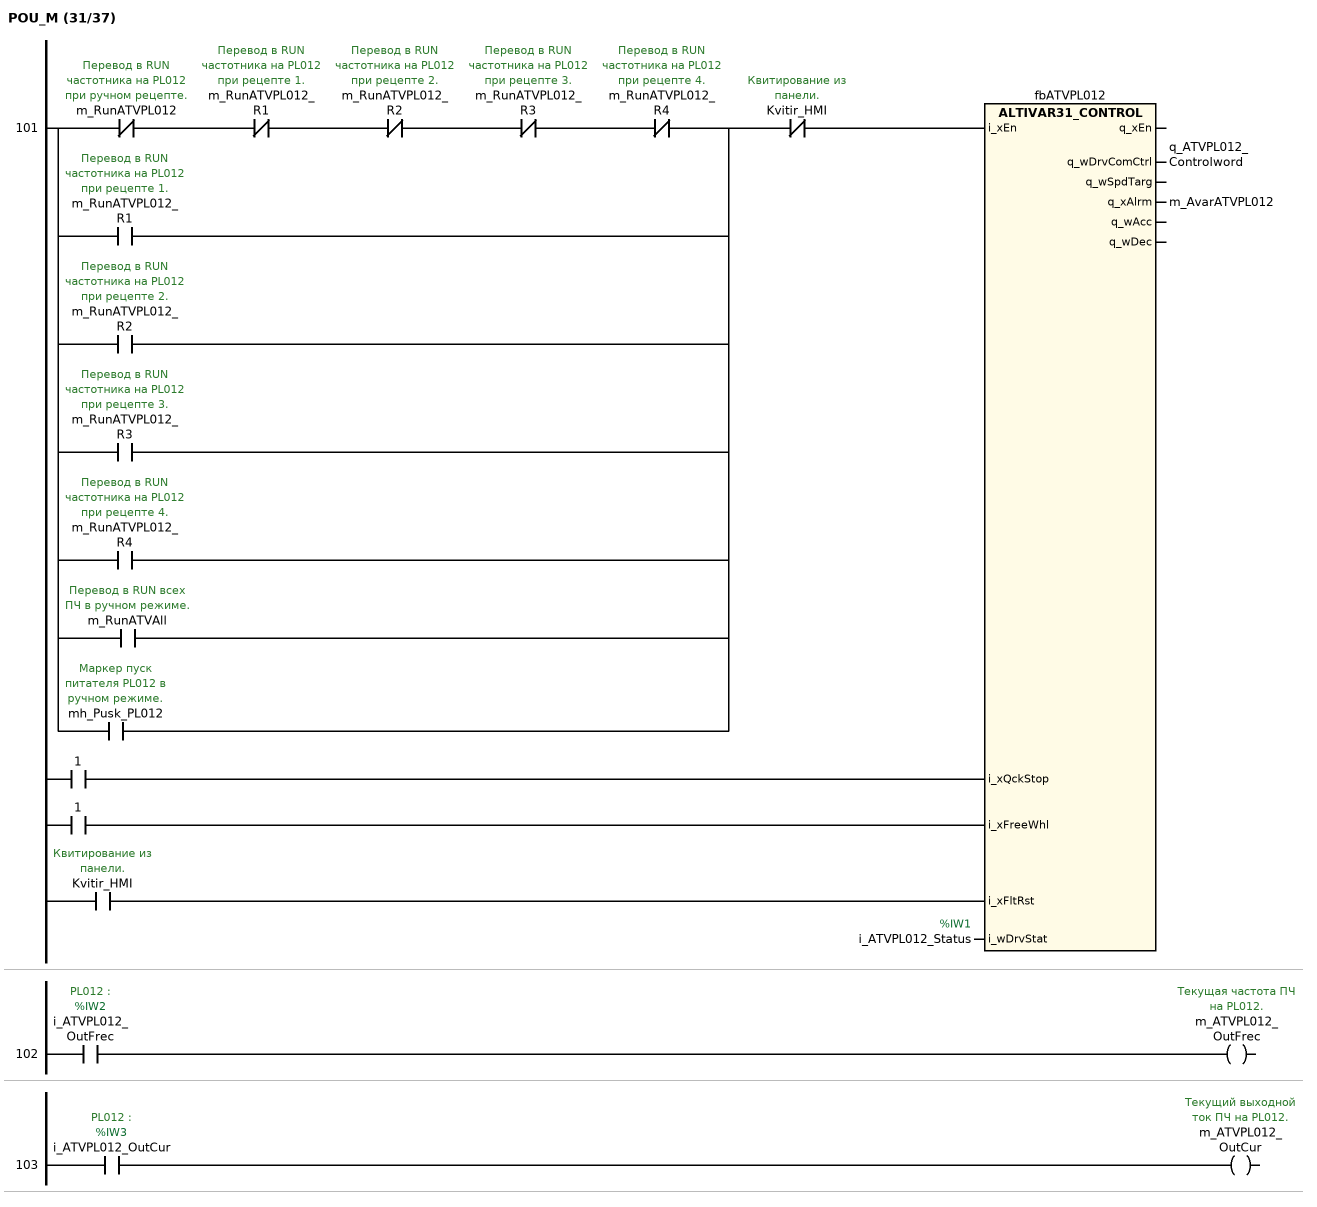
// NETWORK 101
//   fbATVPL012: Блок частотника PL012.
//   m_RunATVPL012: Перевод в RUN частотника на PL012 при ручном рецепте.
//   m_RunATVPL012_R1: Перевод в RUN частотника на PL012 при рецепте 1.
//   m_RunATVPL012_R2: Перевод в RUN частотника на PL012 при рецепте 2.
//   m_RunATVPL012_R3: Перевод в RUN частотника на PL012 при рецепте 3.
//   m_RunATVPL012_R4: Перевод в RUN частотника на PL012 при рецепте 4.
//   m_RunATVAll: Перевод в RUN всех ПЧ в ручном режиме.
//   mh_Pusk_PL012: Маркер пуск питателя PL012 в ручном режиме.
//   Kvitir_HMI: Квитирование из панели.
//   i_ATVPL012_Status: PL012 : | AT %IW1
//   q_ATVPL012_Controlword: PL012 : | AT %QW1
//   m_AvarATVPL012: Ошибка от ПЧ PL012.
fbATVPL012(
    i_xEn := (NOT m_RunATVPL012 AND NOT m_RunATVPL012_R1 AND NOT m_RunATVPL012_R2 AND NOT m_RunATVPL012_R3 AND NOT m_RunATVPL012_R4 OR m_RunATVPL012_R1 OR m_RunATVPL012_R2 OR m_RunATVPL012_R3 OR m_RunATVPL012_R4 OR m_RunATVAll OR mh_Pusk_PL012) AND NOT Kvitir_HMI,
    i_xQckStop := 1,
    i_xFreeWhl := 1,
    i_xFltRst := Kvitir_HMI,
    i_wDrvStat := i_ATVPL012_Status,
    q_wDrvComCtrl => q_ATVPL012_Controlword,
    q_xAlrm => m_AvarATVPL012); // ALTIVAR31_CONTROL

// NETWORK 102
//   i_ATVPL012_OutFrec: PL012 : | AT %IW2
//   m_ATVPL012_OutFrec: Текущая частота ПЧ на PL012.
m_ATVPL012_OutFrec := i_ATVPL012_OutFrec;

// NETWORK 103
//   i_ATVPL012_OutCur: PL012 : | AT %IW3
//   m_ATVPL012_OutCur: Текущий выходной ток ПЧ на PL012.
m_ATVPL012_OutCur := i_ATVPL012_OutCur;

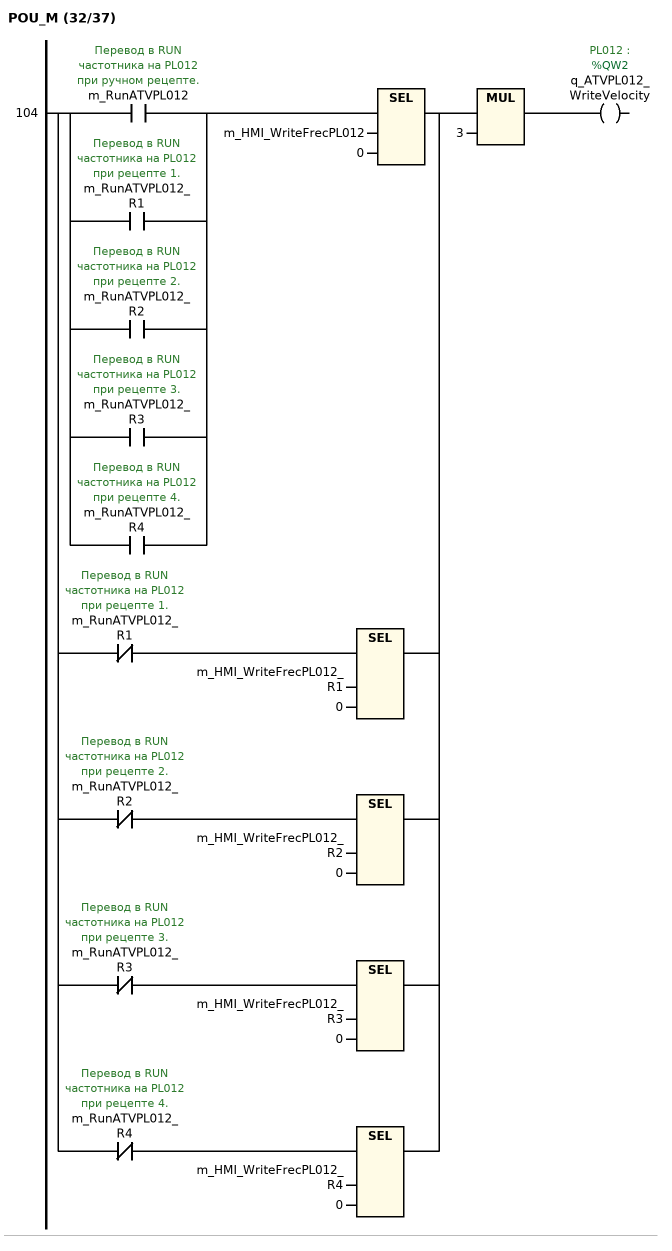
// NETWORK 104
//   m_RunATVPL012: Перевод в RUN частотника на PL012 при ручном рецепте.
//   m_RunATVPL012_R1: Перевод в RUN частотника на PL012 при рецепте 1.
//   m_RunATVPL012_R2: Перевод в RUN частотника на PL012 при рецепте 2.
//   m_RunATVPL012_R3: Перевод в RUN частотника на PL012 при рецепте 3.
//   m_RunATVPL012_R4: Перевод в RUN частотника на PL012 при рецепте 4.
//   m_HMI_WriteFrecPL012: Задание частоты ПЧ на PL012 при ручном рецепте.
//   m_HMI_WriteFrecPL012_R1: Задание частоты ПЧ на PL012 при рецепте 1.
//   m_HMI_WriteFrecPL012_R2: Задание частоты ПЧ на PL012 при рецепте 2.
//   m_HMI_WriteFrecPL012_R3: Задание частоты ПЧ на PL012 при рецепте 3.
//   m_HMI_WriteFrecPL012_R4: Задание частоты ПЧ на PL012 при рецепте 4.
//   q_ATVPL012_WriteVelocity: PL012 : | AT %QW2
q_ATVPL012_WriteVelocity := (SEL(m_RunATVPL012 OR m_RunATVPL012_R1 OR m_RunATVPL012_R2 OR m_RunATVPL012_R3 OR m_RunATVPL012_R4, m_HMI_WriteFrecPL012, 0) OR SEL(NOT m_RunATVPL012_R1, m_HMI_WriteFrecPL012_R1, 0) OR SEL(NOT m_RunATVPL012_R2, m_HMI_WriteFrecPL012_R2, 0) OR SEL(NOT m_RunATVPL012_R3, m_HMI_WriteFrecPL012_R3, 0) OR SEL(NOT m_RunATVPL012_R4, m_HMI_WriteFrecPL012_R4, 0)) * 3;

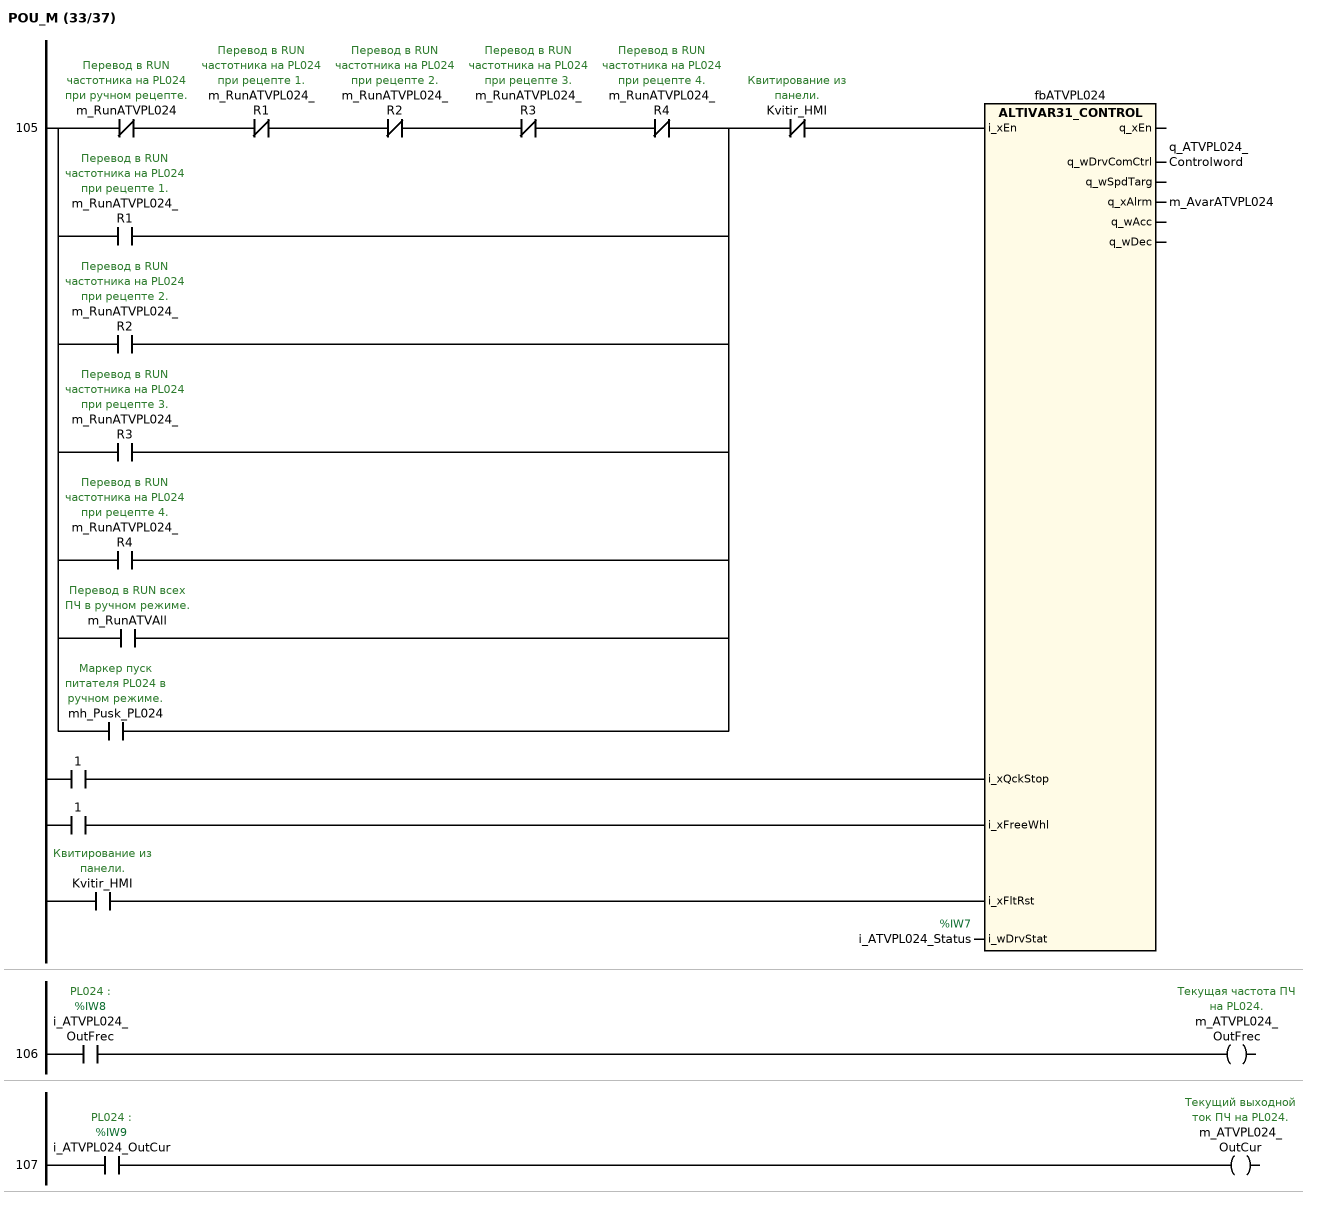
// NETWORK 105
//   fbATVPL024: Блок чатотника PL024.
//   m_RunATVPL024: Перевод в RUN частотника на PL024 при ручном рецепте.
//   m_RunATVPL024_R1: Перевод в RUN частотника на PL024 при рецепте 1.
//   m_RunATVPL024_R2: Перевод в RUN частотника на PL024 при рецепте 2.
//   m_RunATVPL024_R3: Перевод в RUN частотника на PL024 при рецепте 3.
//   m_RunATVPL024_R4: Перевод в RUN частотника на PL024 при рецепте 4.
//   m_RunATVAll: Перевод в RUN всех ПЧ в ручном режиме.
//   mh_Pusk_PL024: Маркер пуск питателя PL024 в ручном режиме.
//   Kvitir_HMI: Квитирование из панели.
//   i_ATVPL024_Status: PL024 : | AT %IW7
//   q_ATVPL024_Controlword: PL024 : | AT %QW5
//   m_AvarATVPL024: Ошибка от ПЧ PL024.
fbATVPL024(
    i_xEn := (NOT m_RunATVPL024 AND NOT m_RunATVPL024_R1 AND NOT m_RunATVPL024_R2 AND NOT m_RunATVPL024_R3 AND NOT m_RunATVPL024_R4 OR m_RunATVPL024_R1 OR m_RunATVPL024_R2 OR m_RunATVPL024_R3 OR m_RunATVPL024_R4 OR m_RunATVAll OR mh_Pusk_PL024) AND NOT Kvitir_HMI,
    i_xQckStop := 1,
    i_xFreeWhl := 1,
    i_xFltRst := Kvitir_HMI,
    i_wDrvStat := i_ATVPL024_Status,
    q_wDrvComCtrl => q_ATVPL024_Controlword,
    q_xAlrm => m_AvarATVPL024); // ALTIVAR31_CONTROL

// NETWORK 106
//   i_ATVPL024_OutFrec: PL024 : | AT %IW8
//   m_ATVPL024_OutFrec: Текущая частота ПЧ на PL024.
m_ATVPL024_OutFrec := i_ATVPL024_OutFrec;

// NETWORK 107
//   i_ATVPL024_OutCur: PL024 : | AT %IW9
//   m_ATVPL024_OutCur: Текущий выходной ток ПЧ на PL024.
m_ATVPL024_OutCur := i_ATVPL024_OutCur;

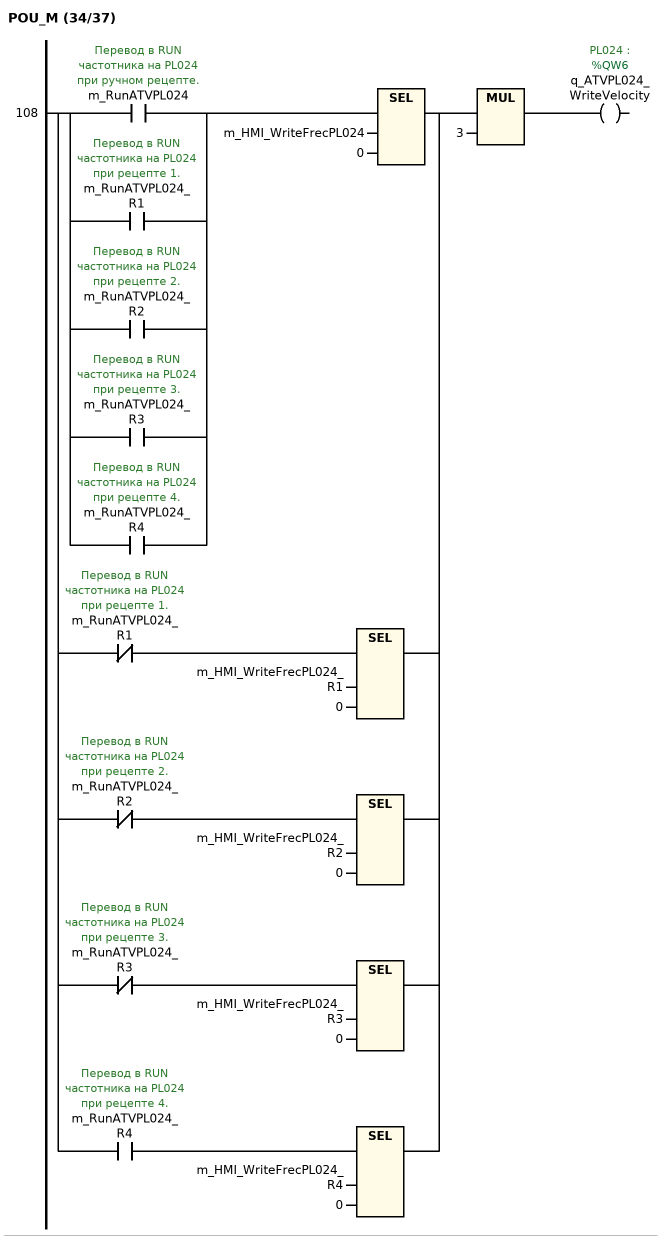
// NETWORK 108
//   m_RunATVPL024: Перевод в RUN частотника на PL024 при ручном рецепте.
//   m_RunATVPL024_R1: Перевод в RUN частотника на PL024 при рецепте 1.
//   m_RunATVPL024_R2: Перевод в RUN частотника на PL024 при рецепте 2.
//   m_RunATVPL024_R3: Перевод в RUN частотника на PL024 при рецепте 3.
//   m_RunATVPL024_R4: Перевод в RUN частотника на PL024 при рецепте 4.
//   m_HMI_WriteFrecPL024: Задание частоты ПЧ на PL024 при ручном рецепте.
//   m_HMI_WriteFrecPL024_R1: Задание частоты ПЧ на PL024 при рецепте 1.
//   m_HMI_WriteFrecPL024_R2: Задание частоты ПЧ на PL024 при рецепте 2.
//   m_HMI_WriteFrecPL024_R3: Задание частоты ПЧ на PL024 при рецепте 3.
//   m_HMI_WriteFrecPL024_R4: Задание частоты ПЧ на PL024 при рецепте 4.
//   q_ATVPL024_WriteVelocity: PL024 : | AT %QW6
q_ATVPL024_WriteVelocity := (SEL(m_RunATVPL024 OR m_RunATVPL024_R1 OR m_RunATVPL024_R2 OR m_RunATVPL024_R3 OR m_RunATVPL024_R4, m_HMI_WriteFrecPL024, 0) OR SEL(NOT m_RunATVPL024_R1, m_HMI_WriteFrecPL024_R1, 0) OR SEL(NOT m_RunATVPL024_R2, m_HMI_WriteFrecPL024_R2, 0) OR SEL(NOT m_RunATVPL024_R3, m_HMI_WriteFrecPL024_R3, 0) OR SEL(m_RunATVPL024_R4, m_HMI_WriteFrecPL024_R4, 0)) * 3;

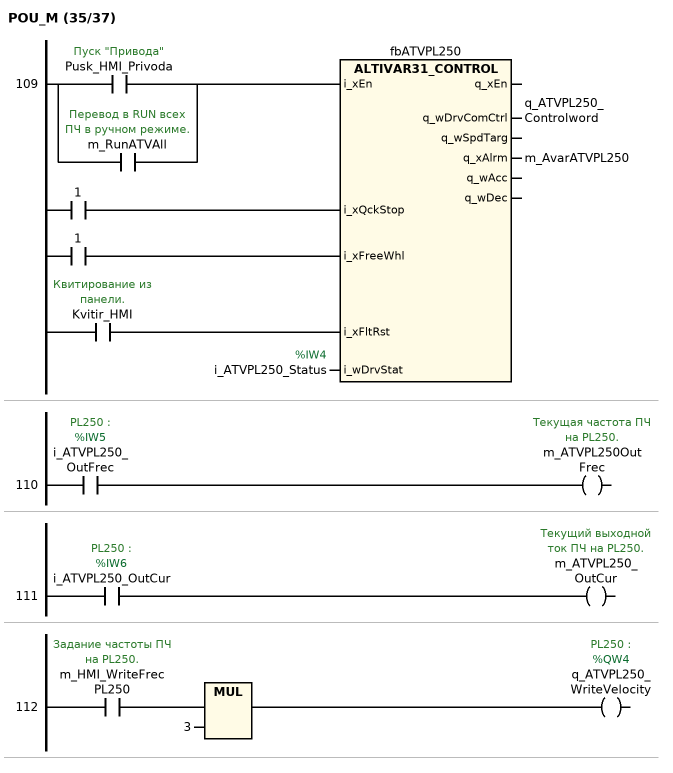
// NETWORK 109
//   fbATVPL250: Блок частотника на PL250.
//   Pusk_HMI_Privoda: Пуск "Привода"
//   m_RunATVAll: Перевод в RUN всех ПЧ в ручном режиме.
//   Kvitir_HMI: Квитирование из панели.
//   i_ATVPL250_Status: PL250 : | AT %IW4
//   q_ATVPL250_Controlword: PL250 : | AT %QW3
//   m_AvarATVPL250: Ошибка от ПЧ PL250.
fbATVPL250(
    i_xEn := Pusk_HMI_Privoda OR m_RunATVAll,
    i_xQckStop := 1,
    i_xFreeWhl := 1,
    i_xFltRst := Kvitir_HMI,
    i_wDrvStat := i_ATVPL250_Status,
    q_wDrvComCtrl => q_ATVPL250_Controlword,
    q_xAlrm => m_AvarATVPL250); // ALTIVAR31_CONTROL

// NETWORK 110
//   i_ATVPL250_OutFrec: PL250 : | AT %IW5
//   m_ATVPL250OutFrec: Текущая частота ПЧ на PL250.
m_ATVPL250OutFrec := i_ATVPL250_OutFrec;

// NETWORK 111
//   i_ATVPL250_OutCur: PL250 : | AT %IW6
//   m_ATVPL250_OutCur: Текущий выходной ток ПЧ на PL250.
m_ATVPL250_OutCur := i_ATVPL250_OutCur;

// NETWORK 112
//   m_HMI_WriteFrecPL250: Задание частоты ПЧ на PL250.
//   q_ATVPL250_WriteVelocity: PL250 : | AT %QW4
q_ATVPL250_WriteVelocity := m_HMI_WriteFrecPL250 * 3;

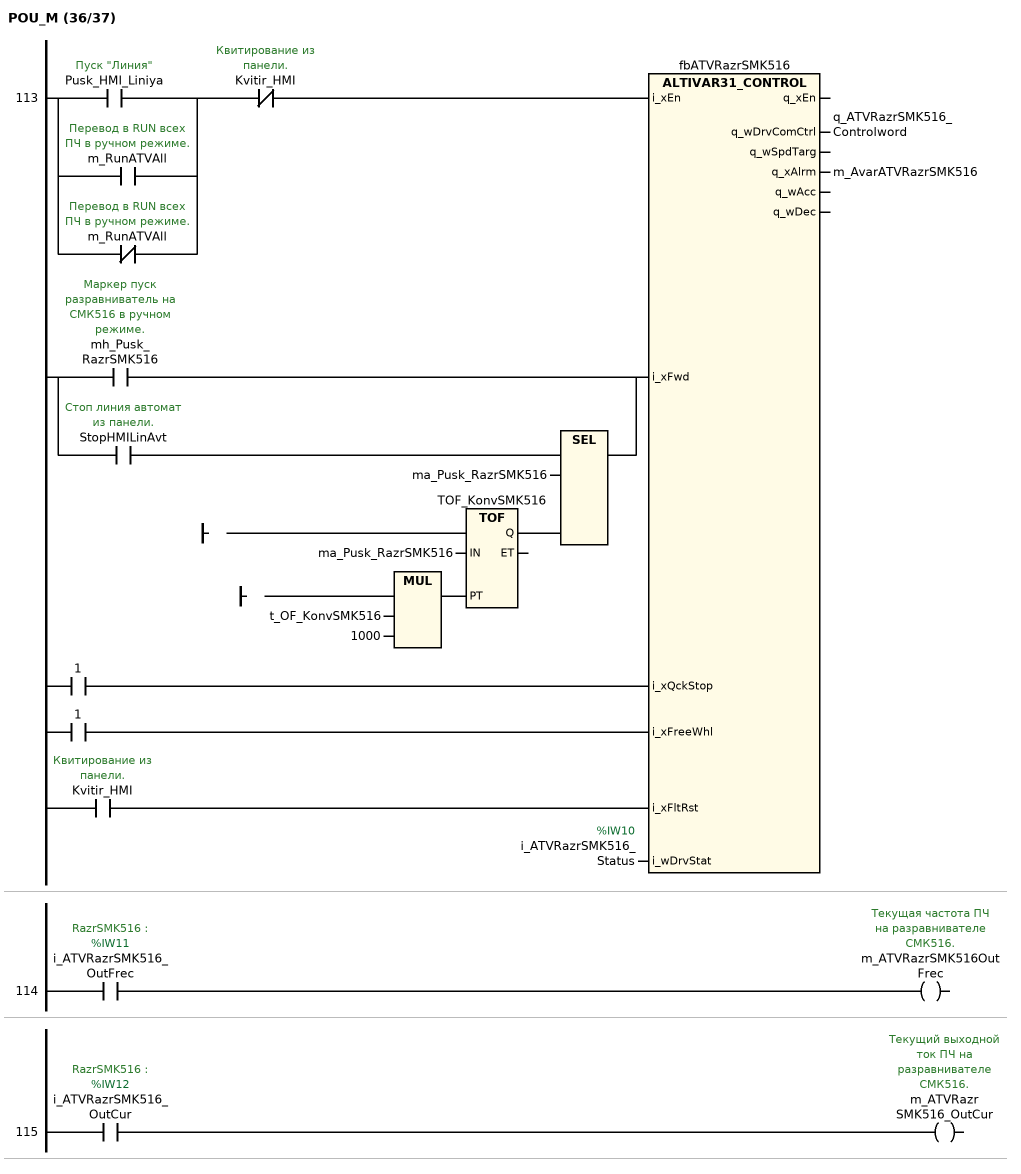
// NETWORK 113
//   fbATVRazrSMK516: Блок частотника на разравнивателе СМК516.
//   Pusk_HMI_Liniya: Пуск "Линия"
//   m_RunATVAll: Перевод в RUN всех ПЧ в ручном режиме.
//   Kvitir_HMI: Квитирование из панели.
//   mh_Pusk_RazrSMK516: Маркер пуск разравниватель на СМК516 в ручном режиме.
//   StopHMILinAvt: Стоп линия автомат из панели.
//   ma_Pusk_RazrSMK516: Маркер пуск разравниватель на СМК516 в автоматическом режиме.
//   TOF_KonvSMK516: Задержка перед выключением конвейера на СМК516 при "Стоп линия автомат".
//   t_OF_KonvSMK516: Время задержки перед выключением конвейера на СМК516 при Стоп Линия Автомат.
//   i_ATVRazrSMK516_Status: RazrSMK516 : | AT %IW10
//   q_ATVRazrSMK516_Controlword: RazrSMK516 : | AT %QW7
//   m_AvarATVRazrSMK516: Ошибка от ПЧ разравнивателя на СМК516.
TOF_KonvSMK516(IN := ma_Pusk_RazrSMK516, PT := t_OF_KonvSMK516 * 1000); // TOF
fbATVRazrSMK516(
    i_xEn := (Pusk_HMI_Liniya OR m_RunATVAll OR NOT m_RunATVAll) AND NOT Kvitir_HMI,
    i_xFwd := mh_Pusk_RazrSMK516 OR SEL(StopHMILinAvt, ma_Pusk_RazrSMK516, TOF_KonvSMK516.Q),
    i_xQckStop := 1,
    i_xFreeWhl := 1,
    i_xFltRst := Kvitir_HMI,
    i_wDrvStat := i_ATVRazrSMK516_Status,
    q_wDrvComCtrl => q_ATVRazrSMK516_Controlword,
    q_xAlrm => m_AvarATVRazrSMK516); // ALTIVAR31_CONTROL

// NETWORK 114
//   i_ATVRazrSMK516_OutFrec: RazrSMK516 : | AT %IW11
//   m_ATVRazrSMK516OutFrec: Текущая частота ПЧ на разравнивателе СМК516.
m_ATVRazrSMK516OutFrec := i_ATVRazrSMK516_OutFrec;

// NETWORK 115
//   i_ATVRazrSMK516_OutCur: RazrSMK516 : | AT %IW12
//   m_ATVRazrSMK516_OutCur: Текущий выходной ток ПЧ на разравнивателе СМК516.
m_ATVRazrSMK516_OutCur := i_ATVRazrSMK516_OutCur;

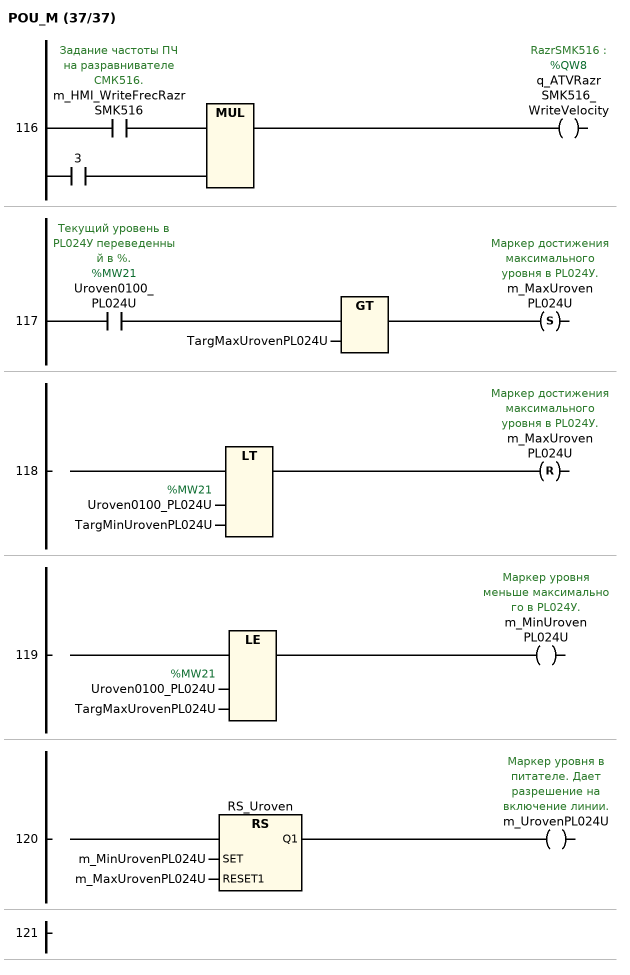
// NETWORK 116
//   m_HMI_WriteFrecRazrSMK516: Задание частоты ПЧ на разравнивателе СМК516.
//   q_ATVRazrSMK516_WriteVelocity: RazrSMK516 : | AT %QW8
q_ATVRazrSMK516_WriteVelocity := m_HMI_WriteFrecRazrSMK516 * 3;

// NETWORK 117
//   Uroven0100_PL024U: Текущий уровень в PL024У переведенный в %. | AT %MW21
//   TargMaxUrovenPL024U: Задание максимально допустимого уровня в PL024У.
//   m_MaxUrovenPL024U: Маркер достижения максимального уровня в PL024У.
m_MaxUrovenPL024U S= Uroven0100_PL024U > TargMaxUrovenPL024U;

// NETWORK 118
//   Uroven0100_PL024U: Текущий уровень в PL024У переведенный в %. | AT %MW21
//   TargMinUrovenPL024U: Задание минимально допустимого уровня в PL024У.
//   m_MaxUrovenPL024U: Маркер достижения максимального уровня в PL024У.
m_MaxUrovenPL024U R= Uroven0100_PL024U < TargMinUrovenPL024U;

// NETWORK 119
//   Uroven0100_PL024U: Текущий уровень в PL024У переведенный в %. | AT %MW21
//   TargMaxUrovenPL024U: Задание максимально допустимого уровня в PL024У.
//   m_MinUrovenPL024U: Маркер уровня меньше максимального в PL024У.
m_MinUrovenPL024U := Uroven0100_PL024U <= TargMaxUrovenPL024U;

// NETWORK 120
//   RS_Uroven: RS-триггер уровня.
//   m_MinUrovenPL024U: Маркер уровня меньше максимального в PL024У.
//   m_MaxUrovenPL024U: Маркер достижения максимального уровня в PL024У.
//   m_UrovenPL024U: Маркер уровня в питателе. Дает разрешение на включение линии.
RS_Uroven(SET := m_MinUrovenPL024U, RESET1 := m_MaxUrovenPL024U); // RS
m_UrovenPL024U := RS_Uroven.Q1;

// NETWORK 121

END_PROGRAM

// MASSA/Application/VisualizationM
